DATA_BLOCK "LBP_SentronPac"   // DB1001
TITLE = SENTRON PAC
{ S7_Optimized_Access := 'FALSE'; DB_Accessible_From_OPC_UA := 'FALSE' }
AUTHOR : SINUMERIK
FAMILY : SINUMERIK_ONE
VERSION : 6.24
// Interface between user program and operating software, contains signals for SENTRON PAC energy monitoring devices / Interface entre programme utilisateur et logiciel d'exploitation, contient des signaux pour unités de surveillance de l'énergie SENTRON PAC
// stored: AutoNumber false, DBAccessibleFromOPCUA false, DBAccessibleFromWebserver false
   VAR RETAIN
      ManualVal { ExternalWritable := 'False'} : Bool;   // Display of manual value / Affichage de la valeur manuelle
      SentronPacMach { ExternalWritable := 'False'} : Bool;   // Sentron PAC represented machine / Machine représentée par Sentron PAC
      FeedInEnergyReadSP { ExternalWritable := 'False'} : Bool;   // Feed-in energy read from Sentron PAC / Énergie alimentée mesurée par Sentron PAC
      FeedBackEnergyReadSP { ExternalWritable := 'False'} : Bool;   // Feed back energy read from Sentron PAC / Énergie réinjectée mesurée par Sentron PAC
      FeedInEnergyReadAuxil { ExternalWritable := 'False'} : Bool;   // Feed-in energy read auxiliary / Énergie alimentée, mesurée par AUX
      FeedBackEnergyReadAuxil { ExternalWritable := 'False'} : Bool;   // Feed back energy read auxiliary / Énergie réinjectée, mesurée par AUX
      res0_6 { ExternalWritable := 'False'} : Bool;   // Reserved / Réservé
      res0_7 { ExternalWritable := 'False'} : Bool;   // Reserved / Réservé
      MeasAuto { ExternalWritable := 'False'} : Bool;   // Measurement by PLC basic program / Mesure par programme de base AP
      res1_1 { ExternalWritable := 'False'} : Bool;   // Reserved / Réservé
      res1_2 { ExternalWritable := 'False'} : Bool;   // Reserved / Réservé
      res1_3 { ExternalWritable := 'False'} : Bool;   // Reserved / Réservé
      res1_4 { ExternalWritable := 'False'} : Bool;   // Reserved / Réservé
      res1_5 { ExternalWritable := 'False'} : Bool;   // Reserved / Réservé
      res1_6 { ExternalWritable := 'False'} : Bool;   // Reserved / Réservé
      res1_7 { ExternalWritable := 'False'} : Bool;   // Reserved / Réservé
      MeasAct : Bool;   // HMI -> PLC: Active measurement / IHM->AP : Mesure active
      res2_1 { ExternalWritable := 'False'} : Bool;   // Reserved / Réservé
      res2_2 { ExternalWritable := 'False'} : Bool;   // Reserved / Réservé
      res2_3 { ExternalWritable := 'False'} : Bool;   // Reserved / Réservé
      res2_4 { ExternalWritable := 'False'} : Bool;   // Reserved / Réservé
      res2_5 { ExternalWritable := 'False'} : Bool;   // Reserved / Réservé
      res2_6 { ExternalWritable := 'False'} : Bool;   // Reserved / Réservé
      res2_7 { ExternalWritable := 'False'} : Bool;   // Reserved / Réservé
      EStateOn { ExternalWritable := 'False'} : Bool;   // Energy state on / État énergie activé
      res3_1 { ExternalWritable := 'False'} : Bool;   // Reserved / Réservé
      res3_2 { ExternalWritable := 'False'} : Bool;   // Reserved / Réservé
      res3_3 { ExternalWritable := 'False'} : Bool;   // Reserved / Réservé
      res3_4 { ExternalWritable := 'False'} : Bool;   // Reserved / Réservé
      res3_5 { ExternalWritable := 'False'} : Bool;   // Reserved / Réservé
      res3_6 { ExternalWritable := 'False'} : Bool;   // Reserved / Réservé
      res3_7 { ExternalWritable := 'False'} : Bool;   // Reserved / Réservé
      ManualValue { ExternalWritable := 'False'} : Real;   // Manual value / Valeur manuelle
      ActivePowerItem { ExternalWritable := 'False'} : Real;   // Active power item / Puissance active position
      ActiveEnergyItem { ExternalWritable := 'False'} : Real;   // Active energy item / Énergie active position
      ReactiveEnergyItem { ExternalWritable := 'False'} : Real;   // Reactive energy item / Énergie réactive position
      ActivePowerSentron { ExternalWritable := 'False'} : Real;   // Active power from Sentron / Puissance active par Sentron
      ActiveEnergySentron { ExternalWritable := 'False'} : Real;   // Active energy from Sentron / Énergie active par Sentron
      ReactiveEnergySentron { ExternalWritable := 'False'} : Real;   // Reactive energy from Sentron / Énergie réactive par Sentron
      ActiveEnergyDay { ExternalWritable := 'False'} : Real;   // Active energy day / Énergie active jour
      ReactiveEnergyDay { ExternalWritable := 'False'} : Real;   // Reactive energy day / Énergie réactive jour
      ActiveEnergyPrevDay { ExternalWritable := 'False'} : Real;   // Active energy previous day / Énergie active jour précédent
      ReactiveEnergyPrevDay { ExternalWritable := 'False'} : Real;   // Reactive energy previous day / Énergie réactive jour précédent
      ActiveEnergyMonth { ExternalWritable := 'False'} : Real;   // Active energy month / Énergie active mois
      ReactiveEnergyMonth { ExternalWritable := 'False'} : Real;   // Reactive energy month / Énergie réactive mois
      ActiveEnergyPrevMonth { ExternalWritable := 'False'} : Real;   // Active energy previous month / Énergie active mois précédent
      ReactiveEnergyPrevMonth { ExternalWritable := 'False'} : Real;   // Reactive energy previous month / Énergie réactive mois précédent
      ActiveEnergyYear { ExternalWritable := 'False'} : Real;   // Active energy year / Énergie active année
      ReactiveEnergyYear { ExternalWritable := 'False'} : Real;   // Reactive energy year / Énergie réactive année
      ActiveEnergyPrevYear { ExternalWritable := 'False'} : Real;   // Active energy previous year / Énergie active année précédente
      ReactiveEnergyPrevYear { ExternalWritable := 'False'} : Real;   // Reactive energy previous year / Énergie réactive année précédente
      res80 { ExternalWritable := 'False'} : Byte;   // Reserved / Réservé
      res81 { ExternalWritable := 'False'} : Byte;   // Reserved / Réservé
      res82 { ExternalWritable := 'False'} : Byte;   // Reserved / Réservé
      res83 { ExternalWritable := 'False'} : Byte;   // Reserved / Réservé
      res84 { ExternalWritable := 'False'} : Byte;   // Reserved / Réservé
      res85 { ExternalWritable := 'False'} : Byte;   // Reserved / Réservé
      res86 { ExternalWritable := 'False'} : Byte;   // Reserved / Réservé
      res87 { ExternalWritable := 'False'} : Byte;   // Reserved / Réservé
      res88 { ExternalWritable := 'False'} : Real;   // Reserved / Réservé
      res92 { ExternalWritable := 'False'} : Real;   // Reserved / Réservé
      ProductionAct { ExternalWritable := 'False'} : Byte;
      ErrDBD20_NAN { ExternalWritable := 'False'} : Bool;   // DBD20: invalid (not a number) / DBD20 : non valide (pas un nombre)
      ErrDBD24_NAN { ExternalWritable := 'False'} : Bool;   // DBD24: invalid (not a number) / DBD24 : non valide (pas un nombre)
      ErrDBD28_NAN { ExternalWritable := 'False'} : Bool;   // DBD28: invalid (not a number) / DBD28 : non valide (pas un nombre)
      res97_3 { ExternalWritable := 'False'} : Bool;   // Reserved / Réservé
      res97_4 { ExternalWritable := 'False'} : Bool;   // Reserved / Réservé
      res97_5 { ExternalWritable := 'False'} : Bool;   // Reserved / Réservé
      res97_6 { ExternalWritable := 'False'} : Bool;   // Reserved / Réservé
      res97_7 { ExternalWritable := 'False'} : Bool;   // Reserved / Réservé
      ErrDBD104_NAN { ExternalWritable := 'False'} : Bool;   // DBD104: invalid (not a number) / DBD104 : non valide (pas un nombre)
      ErrDBD144_NAN { ExternalWritable := 'False'} : Bool;   // DBD144: invalid (not a number) / DBD144 : non valide (pas un nombre)
      ErrDBD184_NAN { ExternalWritable := 'False'} : Bool;   // DBD184: invalid (not a number) / DBD184 : non valide (pas un nombre)
      ErrDBD224_NAN { ExternalWritable := 'False'} : Bool;   // DBD224: invalid (not a number) / DBD224 : non valide (pas un nombre)
      ErrDBD264_NAN { ExternalWritable := 'False'} : Bool;   // DBD264: invalid (not a number) / DBD264 : non valide (pas un nombre)
      ErrDBD304_NAN { ExternalWritable := 'False'} : Bool;   // DBD304: invalid (not a number) / DBD304 : non valide (pas un nombre)
      ErrDBD344_NAN { ExternalWritable := 'False'} : Bool;   // DBD344: invalid (not a number) / DBD344 : non valide (pas un nombre)
      ErrDBD384_NAN { ExternalWritable := 'False'} : Bool;   // DBD384: invalid (not a number) / DBD384 : non valide (pas un nombre)
      ErrDBD424_NAN { ExternalWritable := 'False'} : Bool;   // DBD424: invalid (not a number) / DBD424 : non valide (pas un nombre)
      ErrDBD464_NAN { ExternalWritable := 'False'} : Bool;   // DBD464: invalid (not a number) / DBD464 : non valide (pas un nombre)
      res99_2 { ExternalWritable := 'False'} : Bool;   // Reserved / Réservé
      res99_3 { ExternalWritable := 'False'} : Bool;   // Reserved / Réservé
      res99_4 { ExternalWritable := 'False'} : Bool;   // Reserved / Réservé
      res99_5 { ExternalWritable := 'False'} : Bool;   // Reserved / Réservé
      res99_6 { ExternalWritable := 'False'} : Bool;   // Reserved / Réservé
      res99_7 { ExternalWritable := 'False'} : Bool;   // Reserved / Réservé
      CtrlE_AuxDevice { ExternalWritable := 'False'} : Array[1..10] of Struct
         ProcessAux : Bool;   // Auxiliary present and to be processed / AUX présent et prêt au traitement
         ReadEnergy : Bool;   // Actual values are refreshed; bit is auto-reset / Les valeurs réelles sont actualisées ; le bit est réinitialisé automatiquement
         MeasAct : Bool;   // Measurement values are computed / Calcul des valeurs de mesure en cours
         MeasMode : Bool;   // Difference of actual values is stored / La différence des valeurs réelles est enregistrée
         InputMode : Bool;   // INPUT "ActivePowerAux" is energy in kWh / INPUT "ActivePowerAux" représente l'énergie en kWh
         res0_5 : Bool;
         res0_6 : Bool;
         ResetAux : Bool;   // Auxiliary data are deleted / Les données AUX sont supprimées
         res1 : Byte;   // Reserved / Réservé
         res2 : Word;   // Reserved / Réservé
         ActivePowerAux : Real;   // [kW]/[kWh] power/energy of auxiliary, written by customer / [kW]/[kWh] puissance/énergie AUX, renseignée par le client
         ActiveEnAux : Real;   // [kWh] actual value of fed-in-energy / [kWh] valeur réelle de l'énergie consommée
         ReActiveEnAux : Real;   // [kWh] actual value of fed-back energy / [kWh] valeur réelle de l'énergie réinjectée
         ActiveEnAuxMeasON : Real;   // [kWh] value of fed-in-energy at start of measurement / [kWh] valeur réelle de l'énergie consommée au début de la mesure
         ReActiveEnAuxMeasON : Real;   // [kWh] value of fed-back energy at start of measurement / Wh] valeur réelle de l'énergie réinjectée au début de la mesure
         ActiveEnAuxMeasOFF : Real;   // [kWh] value of fed-in-energy at end of measurement / [kWh] valeur réelle de l'énergie consommée à la fin de la mesure
         ReActiveEnAuxMeasOFF : Real;   // [kWh] value of fed-back energy at end of measurement / [kWh] valeur réelle de l'énergie réinjectée à la fin de la mesure
         res32 : DWord;   // Reserved / Réservé
         res36 : Real;   // Reserved / Réservé
      END_STRUCT;
   END_VAR
BEGIN
   // CtrlE_AuxDevice[2].ProcessAux : Auxiliary present and to be processed / AUX présent et prêt au traitement
   // CtrlE_AuxDevice[3].ProcessAux : Auxiliary present and to be processed / AUX présent et prêt au traitement
   // CtrlE_AuxDevice[4].ProcessAux : Auxiliary present and to be processed / AUX présent et prêt au traitement
   // CtrlE_AuxDevice[5].ProcessAux : Auxiliary present and to be processed / AUX présent et prêt au traitement
   // CtrlE_AuxDevice[6].ProcessAux : Auxiliary present and to be processed / AUX présent et prêt au traitement
   // CtrlE_AuxDevice[7].ProcessAux : Auxiliary present and to be processed / AUX présent et prêt au traitement
   // CtrlE_AuxDevice[8].ProcessAux : Auxiliary present and to be processed / AUX présent et prêt au traitement
   // CtrlE_AuxDevice[9].ProcessAux : Auxiliary present and to be processed / AUX présent et prêt au traitement
   // CtrlE_AuxDevice[10].ProcessAux : Auxiliary present and to be processed / AUX présent et prêt au traitement
   // CtrlE_AuxDevice[2].ReadEnergy : Actual values are refreshed; bit is auto-reset / Les valeurs réelles sont actualisées ; le bit est réinitialisé automatiquement
   // CtrlE_AuxDevice[3].ReadEnergy : Actual values are refreshed; bit is auto-reset / Les valeurs réelles sont actualisées ; le bit est réinitialisé automatiquement
   // CtrlE_AuxDevice[4].ReadEnergy : Actual values are refreshed; bit is auto-reset / Les valeurs réelles sont actualisées ; le bit est réinitialisé automatiquement
   // CtrlE_AuxDevice[5].ReadEnergy : Actual values are refreshed; bit is auto-reset / Les valeurs réelles sont actualisées ; le bit est réinitialisé automatiquement
   // CtrlE_AuxDevice[6].ReadEnergy : Actual values are refreshed; bit is auto-reset / Les valeurs réelles sont actualisées ; le bit est réinitialisé automatiquement
   // CtrlE_AuxDevice[7].ReadEnergy : Actual values are refreshed; bit is auto-reset / Les valeurs réelles sont actualisées ; le bit est réinitialisé automatiquement
   // CtrlE_AuxDevice[8].ReadEnergy : Actual values are refreshed; bit is auto-reset / Les valeurs réelles sont actualisées ; le bit est réinitialisé automatiquement
   // CtrlE_AuxDevice[9].ReadEnergy : Actual values are refreshed; bit is auto-reset / Les valeurs réelles sont actualisées ; le bit est réinitialisé automatiquement
   // CtrlE_AuxDevice[10].ReadEnergy : Actual values are refreshed; bit is auto-reset / Les valeurs réelles sont actualisées ; le bit est réinitialisé automatiquement
   // CtrlE_AuxDevice[2].MeasAct : Measurement values are computed / Calcul des valeurs de mesure en cours
   // CtrlE_AuxDevice[3].MeasAct : Measurement values are computed / Calcul des valeurs de mesure en cours
   // CtrlE_AuxDevice[4].MeasAct : Measurement values are computed / Calcul des valeurs de mesure en cours
   // CtrlE_AuxDevice[5].MeasAct : Measurement values are computed / Calcul des valeurs de mesure en cours
   // CtrlE_AuxDevice[6].MeasAct : Measurement values are computed / Calcul des valeurs de mesure en cours
   // CtrlE_AuxDevice[7].MeasAct : Measurement values are computed / Calcul des valeurs de mesure en cours
   // CtrlE_AuxDevice[8].MeasAct : Measurement values are computed / Calcul des valeurs de mesure en cours
   // CtrlE_AuxDevice[9].MeasAct : Measurement values are computed / Calcul des valeurs de mesure en cours
   // CtrlE_AuxDevice[10].MeasAct : Measurement values are computed / Calcul des valeurs de mesure en cours
   // CtrlE_AuxDevice[2].MeasMode : Difference of actual values is stored / La différence des valeurs réelles est enregistrée
   // CtrlE_AuxDevice[3].MeasMode : Difference of actual values is stored / La différence des valeurs réelles est enregistrée
   // CtrlE_AuxDevice[4].MeasMode : Difference of actual values is stored / La différence des valeurs réelles est enregistrée
   // CtrlE_AuxDevice[5].MeasMode : Difference of actual values is stored / La différence des valeurs réelles est enregistrée
   // CtrlE_AuxDevice[6].MeasMode : Difference of actual values is stored / La différence des valeurs réelles est enregistrée
   // CtrlE_AuxDevice[7].MeasMode : Difference of actual values is stored / La différence des valeurs réelles est enregistrée
   // CtrlE_AuxDevice[8].MeasMode : Difference of actual values is stored / La différence des valeurs réelles est enregistrée
   // CtrlE_AuxDevice[9].MeasMode : Difference of actual values is stored / La différence des valeurs réelles est enregistrée
   // CtrlE_AuxDevice[10].MeasMode : Difference of actual values is stored / La différence des valeurs réelles est enregistrée
   // CtrlE_AuxDevice[2].InputMode : INPUT "ActivePowerAux" is energy in kWh / INPUT "ActivePowerAux" représente l'énergie en kWh
   // CtrlE_AuxDevice[3].InputMode : INPUT "ActivePowerAux" is energy in kWh / INPUT "ActivePowerAux" représente l'énergie en kWh
   // CtrlE_AuxDevice[4].InputMode : INPUT "ActivePowerAux" is energy in kWh / INPUT "ActivePowerAux" représente l'énergie en kWh
   // CtrlE_AuxDevice[5].InputMode : INPUT "ActivePowerAux" is energy in kWh / INPUT "ActivePowerAux" représente l'énergie en kWh
   // CtrlE_AuxDevice[6].InputMode : INPUT "ActivePowerAux" is energy in kWh / INPUT "ActivePowerAux" représente l'énergie en kWh
   // CtrlE_AuxDevice[7].InputMode : INPUT "ActivePowerAux" is energy in kWh / INPUT "ActivePowerAux" représente l'énergie en kWh
   // CtrlE_AuxDevice[8].InputMode : INPUT "ActivePowerAux" is energy in kWh / INPUT "ActivePowerAux" représente l'énergie en kWh
   // CtrlE_AuxDevice[9].InputMode : INPUT "ActivePowerAux" is energy in kWh / INPUT "ActivePowerAux" représente l'énergie en kWh
   // CtrlE_AuxDevice[10].InputMode : INPUT "ActivePowerAux" is energy in kWh / INPUT "ActivePowerAux" représente l'énergie en kWh
   // CtrlE_AuxDevice[2].ResetAux : Auxiliary data are deleted / Les données AUX sont supprimées
   // CtrlE_AuxDevice[3].ResetAux : Auxiliary data are deleted / Les données AUX sont supprimées
   // CtrlE_AuxDevice[4].ResetAux : Auxiliary data are deleted / Les données AUX sont supprimées
   // CtrlE_AuxDevice[5].ResetAux : Auxiliary data are deleted / Les données AUX sont supprimées
   // CtrlE_AuxDevice[6].ResetAux : Auxiliary data are deleted / Les données AUX sont supprimées
   // CtrlE_AuxDevice[7].ResetAux : Auxiliary data are deleted / Les données AUX sont supprimées
   // CtrlE_AuxDevice[8].ResetAux : Auxiliary data are deleted / Les données AUX sont supprimées
   // CtrlE_AuxDevice[9].ResetAux : Auxiliary data are deleted / Les données AUX sont supprimées
   // CtrlE_AuxDevice[10].ResetAux : Auxiliary data are deleted / Les données AUX sont supprimées
   // CtrlE_AuxDevice[2].res1 : Reserved / Réservé
   // CtrlE_AuxDevice[3].res1 : Reserved / Réservé
   // CtrlE_AuxDevice[4].res1 : Reserved / Réservé
   // CtrlE_AuxDevice[5].res1 : Reserved / Réservé
   // CtrlE_AuxDevice[6].res1 : Reserved / Réservé
   // CtrlE_AuxDevice[7].res1 : Reserved / Réservé
   // CtrlE_AuxDevice[8].res1 : Reserved / Réservé
   // CtrlE_AuxDevice[9].res1 : Reserved / Réservé
   // CtrlE_AuxDevice[10].res1 : Reserved / Réservé
   // CtrlE_AuxDevice[2].res2 : Reserved / Réservé
   // CtrlE_AuxDevice[3].res2 : Reserved / Réservé
   // CtrlE_AuxDevice[4].res2 : Reserved / Réservé
   // CtrlE_AuxDevice[5].res2 : Reserved / Réservé
   // CtrlE_AuxDevice[6].res2 : Reserved / Réservé
   // CtrlE_AuxDevice[7].res2 : Reserved / Réservé
   // CtrlE_AuxDevice[8].res2 : Reserved / Réservé
   // CtrlE_AuxDevice[9].res2 : Reserved / Réservé
   // CtrlE_AuxDevice[10].res2 : Reserved / Réservé
   // CtrlE_AuxDevice[2].ActivePowerAux : [kW]/[kWh] power/energy of auxiliary, written by customer / [kW]/[kWh] puissance/énergie AUX, renseignée par le client
   // CtrlE_AuxDevice[3].ActivePowerAux : [kW]/[kWh] power/energy of auxiliary, written by customer / [kW]/[kWh] puissance/énergie AUX, renseignée par le client
   // CtrlE_AuxDevice[4].ActivePowerAux : [kW]/[kWh] power/energy of auxiliary, written by customer / [kW]/[kWh] puissance/énergie AUX, renseignée par le client
   // CtrlE_AuxDevice[5].ActivePowerAux : [kW]/[kWh] power/energy of auxiliary, written by customer / [kW]/[kWh] puissance/énergie AUX, renseignée par le client
   // CtrlE_AuxDevice[6].ActivePowerAux : [kW]/[kWh] power/energy of auxiliary, written by customer / [kW]/[kWh] puissance/énergie AUX, renseignée par le client
   // CtrlE_AuxDevice[7].ActivePowerAux : [kW]/[kWh] power/energy of auxiliary, written by customer / [kW]/[kWh] puissance/énergie AUX, renseignée par le client
   // CtrlE_AuxDevice[8].ActivePowerAux : [kW]/[kWh] power/energy of auxiliary, written by customer / [kW]/[kWh] puissance/énergie AUX, renseignée par le client
   // CtrlE_AuxDevice[9].ActivePowerAux : [kW]/[kWh] power/energy of auxiliary, written by customer / [kW]/[kWh] puissance/énergie AUX, renseignée par le client
   // CtrlE_AuxDevice[10].ActivePowerAux : [kW]/[kWh] power/energy of auxiliary, written by customer / [kW]/[kWh] puissance/énergie AUX, renseignée par le client
   // CtrlE_AuxDevice[2].ActiveEnAux : [kWh] actual value of fed-in-energy / [kWh] valeur réelle de l'énergie consommée
   // CtrlE_AuxDevice[3].ActiveEnAux : [kWh] actual value of fed-in-energy / [kWh] valeur réelle de l'énergie consommée
   // CtrlE_AuxDevice[4].ActiveEnAux : [kWh] actual value of fed-in-energy / [kWh] valeur réelle de l'énergie consommée
   // CtrlE_AuxDevice[5].ActiveEnAux : [kWh] actual value of fed-in-energy / [kWh] valeur réelle de l'énergie consommée
   // CtrlE_AuxDevice[6].ActiveEnAux : [kWh] actual value of fed-in-energy / [kWh] valeur réelle de l'énergie consommée
   // CtrlE_AuxDevice[7].ActiveEnAux : [kWh] actual value of fed-in-energy / [kWh] valeur réelle de l'énergie consommée
   // CtrlE_AuxDevice[8].ActiveEnAux : [kWh] actual value of fed-in-energy / [kWh] valeur réelle de l'énergie consommée
   // CtrlE_AuxDevice[9].ActiveEnAux : [kWh] actual value of fed-in-energy / [kWh] valeur réelle de l'énergie consommée
   // CtrlE_AuxDevice[10].ActiveEnAux : [kWh] actual value of fed-in-energy / [kWh] valeur réelle de l'énergie consommée
   // CtrlE_AuxDevice[2].ReActiveEnAux : [kWh] actual value of fed-back energy / [kWh] valeur réelle de l'énergie réinjectée
   // CtrlE_AuxDevice[3].ReActiveEnAux : [kWh] actual value of fed-back energy / [kWh] valeur réelle de l'énergie réinjectée
   // CtrlE_AuxDevice[4].ReActiveEnAux : [kWh] actual value of fed-back energy / [kWh] valeur réelle de l'énergie réinjectée
   // CtrlE_AuxDevice[5].ReActiveEnAux : [kWh] actual value of fed-back energy / [kWh] valeur réelle de l'énergie réinjectée
   // CtrlE_AuxDevice[6].ReActiveEnAux : [kWh] actual value of fed-back energy / [kWh] valeur réelle de l'énergie réinjectée
   // CtrlE_AuxDevice[7].ReActiveEnAux : [kWh] actual value of fed-back energy / [kWh] valeur réelle de l'énergie réinjectée
   // CtrlE_AuxDevice[8].ReActiveEnAux : [kWh] actual value of fed-back energy / [kWh] valeur réelle de l'énergie réinjectée
   // CtrlE_AuxDevice[9].ReActiveEnAux : [kWh] actual value of fed-back energy / [kWh] valeur réelle de l'énergie réinjectée
   // CtrlE_AuxDevice[10].ReActiveEnAux : [kWh] actual value of fed-back energy / [kWh] valeur réelle de l'énergie réinjectée
   // CtrlE_AuxDevice[2].ActiveEnAuxMeasON : [kWh] value of fed-in-energy at start of measurement / [kWh] valeur réelle de l'énergie consommée au début de la mesure
   // CtrlE_AuxDevice[3].ActiveEnAuxMeasON : [kWh] value of fed-in-energy at start of measurement / [kWh] valeur réelle de l'énergie consommée au début de la mesure
   // CtrlE_AuxDevice[4].ActiveEnAuxMeasON : [kWh] value of fed-in-energy at start of measurement / [kWh] valeur réelle de l'énergie consommée au début de la mesure
   // CtrlE_AuxDevice[5].ActiveEnAuxMeasON : [kWh] value of fed-in-energy at start of measurement / [kWh] valeur réelle de l'énergie consommée au début de la mesure
   // CtrlE_AuxDevice[6].ActiveEnAuxMeasON : [kWh] value of fed-in-energy at start of measurement / [kWh] valeur réelle de l'énergie consommée au début de la mesure
   // CtrlE_AuxDevice[7].ActiveEnAuxMeasON : [kWh] value of fed-in-energy at start of measurement / [kWh] valeur réelle de l'énergie consommée au début de la mesure
   // CtrlE_AuxDevice[8].ActiveEnAuxMeasON : [kWh] value of fed-in-energy at start of measurement / [kWh] valeur réelle de l'énergie consommée au début de la mesure
   // CtrlE_AuxDevice[9].ActiveEnAuxMeasON : [kWh] value of fed-in-energy at start of measurement / [kWh] valeur réelle de l'énergie consommée au début de la mesure
   // CtrlE_AuxDevice[10].ActiveEnAuxMeasON : [kWh] value of fed-in-energy at start of measurement / [kWh] valeur réelle de l'énergie consommée au début de la mesure
   // CtrlE_AuxDevice[2].ReActiveEnAuxMeasON : [kWh] value of fed-back energy at start of measurement / Wh] valeur réelle de l'énergie réinjectée au début de la mesure
   // CtrlE_AuxDevice[3].ReActiveEnAuxMeasON : [kWh] value of fed-back energy at start of measurement / Wh] valeur réelle de l'énergie réinjectée au début de la mesure
   // CtrlE_AuxDevice[4].ReActiveEnAuxMeasON : [kWh] value of fed-back energy at start of measurement / Wh] valeur réelle de l'énergie réinjectée au début de la mesure
   // CtrlE_AuxDevice[5].ReActiveEnAuxMeasON : [kWh] value of fed-back energy at start of measurement / Wh] valeur réelle de l'énergie réinjectée au début de la mesure
   // CtrlE_AuxDevice[6].ReActiveEnAuxMeasON : [kWh] value of fed-back energy at start of measurement / Wh] valeur réelle de l'énergie réinjectée au début de la mesure
   // CtrlE_AuxDevice[7].ReActiveEnAuxMeasON : [kWh] value of fed-back energy at start of measurement / Wh] valeur réelle de l'énergie réinjectée au début de la mesure
   // CtrlE_AuxDevice[8].ReActiveEnAuxMeasON : [kWh] value of fed-back energy at start of measurement / Wh] valeur réelle de l'énergie réinjectée au début de la mesure
   // CtrlE_AuxDevice[9].ReActiveEnAuxMeasON : [kWh] value of fed-back energy at start of measurement / Wh] valeur réelle de l'énergie réinjectée au début de la mesure
   // CtrlE_AuxDevice[10].ReActiveEnAuxMeasON : [kWh] value of fed-back energy at start of measurement / Wh] valeur réelle de l'énergie réinjectée au début de la mesure
   // CtrlE_AuxDevice[2].ActiveEnAuxMeasOFF : [kWh] value of fed-in-energy at end of measurement / [kWh] valeur réelle de l'énergie consommée à la fin de la mesure
   // CtrlE_AuxDevice[3].ActiveEnAuxMeasOFF : [kWh] value of fed-in-energy at end of measurement / [kWh] valeur réelle de l'énergie consommée à la fin de la mesure
   // CtrlE_AuxDevice[4].ActiveEnAuxMeasOFF : [kWh] value of fed-in-energy at end of measurement / [kWh] valeur réelle de l'énergie consommée à la fin de la mesure
   // CtrlE_AuxDevice[5].ActiveEnAuxMeasOFF : [kWh] value of fed-in-energy at end of measurement / [kWh] valeur réelle de l'énergie consommée à la fin de la mesure
   // CtrlE_AuxDevice[6].ActiveEnAuxMeasOFF : [kWh] value of fed-in-energy at end of measurement / [kWh] valeur réelle de l'énergie consommée à la fin de la mesure
   // CtrlE_AuxDevice[7].ActiveEnAuxMeasOFF : [kWh] value of fed-in-energy at end of measurement / [kWh] valeur réelle de l'énergie consommée à la fin de la mesure
   // CtrlE_AuxDevice[8].ActiveEnAuxMeasOFF : [kWh] value of fed-in-energy at end of measurement / [kWh] valeur réelle de l'énergie consommée à la fin de la mesure
   // CtrlE_AuxDevice[9].ActiveEnAuxMeasOFF : [kWh] value of fed-in-energy at end of measurement / [kWh] valeur réelle de l'énergie consommée à la fin de la mesure
   // CtrlE_AuxDevice[10].ActiveEnAuxMeasOFF : [kWh] value of fed-in-energy at end of measurement / [kWh] valeur réelle de l'énergie consommée à la fin de la mesure
   // CtrlE_AuxDevice[2].ReActiveEnAuxMeasOFF : [kWh] value of fed-back energy at end of measurement / [kWh] valeur réelle de l'énergie réinjectée à la fin de la mesure
   // CtrlE_AuxDevice[3].ReActiveEnAuxMeasOFF : [kWh] value of fed-back energy at end of measurement / [kWh] valeur réelle de l'énergie réinjectée à la fin de la mesure
   // CtrlE_AuxDevice[4].ReActiveEnAuxMeasOFF : [kWh] value of fed-back energy at end of measurement / [kWh] valeur réelle de l'énergie réinjectée à la fin de la mesure
   // CtrlE_AuxDevice[5].ReActiveEnAuxMeasOFF : [kWh] value of fed-back energy at end of measurement / [kWh] valeur réelle de l'énergie réinjectée à la fin de la mesure
   // CtrlE_AuxDevice[6].ReActiveEnAuxMeasOFF : [kWh] value of fed-back energy at end of measurement / [kWh] valeur réelle de l'énergie réinjectée à la fin de la mesure
   // CtrlE_AuxDevice[7].ReActiveEnAuxMeasOFF : [kWh] value of fed-back energy at end of measurement / [kWh] valeur réelle de l'énergie réinjectée à la fin de la mesure
   // CtrlE_AuxDevice[8].ReActiveEnAuxMeasOFF : [kWh] value of fed-back energy at end of measurement / [kWh] valeur réelle de l'énergie réinjectée à la fin de la mesure
   // CtrlE_AuxDevice[9].ReActiveEnAuxMeasOFF : [kWh] value of fed-back energy at end of measurement / [kWh] valeur réelle de l'énergie réinjectée à la fin de la mesure
   // CtrlE_AuxDevice[10].ReActiveEnAuxMeasOFF : [kWh] value of fed-back energy at end of measurement / [kWh] valeur réelle de l'énergie réinjectée à la fin de la mesure
   // CtrlE_AuxDevice[2].res32 : Reserved / Réservé
   // CtrlE_AuxDevice[3].res32 : Reserved / Réservé
   // CtrlE_AuxDevice[4].res32 : Reserved / Réservé
   // CtrlE_AuxDevice[5].res32 : Reserved / Réservé
   // CtrlE_AuxDevice[6].res32 : Reserved / Réservé
   // CtrlE_AuxDevice[7].res32 : Reserved / Réservé
   // CtrlE_AuxDevice[8].res32 : Reserved / Réservé
   // CtrlE_AuxDevice[9].res32 : Reserved / Réservé
   // CtrlE_AuxDevice[10].res32 : Reserved / Réservé
   // CtrlE_AuxDevice[2].res36 : Reserved / Réservé
   // CtrlE_AuxDevice[3].res36 : Reserved / Réservé
   // CtrlE_AuxDevice[4].res36 : Reserved / Réservé
   // CtrlE_AuxDevice[5].res36 : Reserved / Réservé
   // CtrlE_AuxDevice[6].res36 : Reserved / Réservé
   // CtrlE_AuxDevice[7].res36 : Reserved / Réservé
   // CtrlE_AuxDevice[8].res36 : Reserved / Réservé
   // CtrlE_AuxDevice[9].res36 : Reserved / Réservé
   // CtrlE_AuxDevice[10].res36 : Reserved / Réservé
END_DATA_BLOCK

DATA_BLOCK "LBP_SpindleTempSensor"   // DB1002
TITLE = Spindle temperature sensors / Sondes thermométriques de broche
{ S7_Optimized_Access := 'FALSE' }
AUTHOR : SINUMERIK
FAMILY : SINUMERIK_ONE
VERSION : 6.24
// Interface between user program and operating software, contains signals for spindle temperature sensors / Interface entre programme utilisateur et logiciel d'exploitation, contient des signaux pour sondes thermométriques de broche
// stored: AutoNumber false
   VAR RETAIN
      Sp : Array[1..2] of Struct   // Spindle / Broche
         TS : Array[1..6] of Struct   // Temperature sensor / Sonde thermométrique
            MountPlace : Int;   // Sensor assembly location / Emplacement du module capteur
            Res1 : Int;
            ActVal : Real;   // Temperature sensor actual value [°C] / Sonde thermométrique valeur réelle [°C]
            WarnThreshold : Real;   // Temperature sensor warning threshold value [°C] / Sonde thermométrique valeur seuil d'alarme
            WarnNumLimitViol : Int;   // Number of warning threshold value violations / Nombre de dépassements de la valeur seuil d'alarme
            WarnTsViolYY : Byte;   // Last warning threshold value violation: year / Dernier dépassement de la valeur seuil d'alarme : année
            WarnTsViolMM : Byte;   // Last warning threshold value violation: month / Dernier dépassement de la valeur seuil d'alarme : mois
            WarnTsViolDD : Byte;   // Last warning threshold value violation: day / Dernier dépassement de la valeur seuil d'alarme : jour
            WarnTsViolH : Byte;   // Last warning threshold value violation: hour / Dernier dépassement de la valeur seuil d'alarme : heure
            WarnTsViolM : Byte;   // Last warning threshold value violation: minute / Dernier dépassement de la valeur seuil d'alarme : minute
            WarnTsViolS : Byte;   // Last warning threshold value violation: second / Dernier dépassement de la valeur seuil d'alarme : seconde
            WarnDurLimitViol : DInt;   // Duration of warning threshold value violations / Durée de dépassement de la valeur seuil d'alarme
            FaultThreshold : Real;   // Temperature sensor fault threshold value [°C] / Sonde thermométrique valeur seuil de défaut
            FaultNumLimitViol : Int;   // Number of fault threshold value violations / Nombre de dépassements de la valeur seuil de défaut
            FaultTsViolYY : Byte;   // Last fault threshold value violation: year / Dernier dépassement de la valeur seuil de défaut : année
            FaultTsViolMM : Byte;   // Last fault threshold value violation: month / Dernier dépassement de la valeur seuil de défaut : mois
            FaultTsViolDD : Byte;   // Last fault threshold value violation: day / Dernier dépassement de la valeur seuil de défaut : jour
            FaultTsViolH : Byte;   // Last fault threshold value violation: hour / Dernier dépassement de la valeur seuil de défaut : heure
            FaultTsViolM : Byte;   // Last fault threshold value violation: minute / Dernier dépassement de la valeur seuil de défaut : minute
            FaultTsViolS : Byte;   // Last fault threshold value violation: second / Dernier dépassement de la valeur seuil de défaut : seconde
            FaultDurLimitViol : DInt;   // Duration of fault threshold value violations / Durée de dépassement de la valeur seuil de défaut
         END_STRUCT;
      END_STRUCT;
   END_VAR
BEGIN
   // Sp[1].TS[2].MountPlace : Sensor assembly location / Emplacement du module capteur
   // Sp[1].TS[3].MountPlace : Sensor assembly location / Emplacement du module capteur
   // Sp[1].TS[4].MountPlace : Sensor assembly location / Emplacement du module capteur
   // Sp[1].TS[5].MountPlace : Sensor assembly location / Emplacement du module capteur
   // Sp[1].TS[6].MountPlace : Sensor assembly location / Emplacement du module capteur
   // Sp[2].TS[1].MountPlace : Sensor assembly location / Emplacement du module capteur
   // Sp[2].TS[2].MountPlace : Sensor assembly location / Emplacement du module capteur
   // Sp[2].TS[3].MountPlace : Sensor assembly location / Emplacement du module capteur
   // Sp[2].TS[4].MountPlace : Sensor assembly location / Emplacement du module capteur
   // Sp[2].TS[5].MountPlace : Sensor assembly location / Emplacement du module capteur
   // Sp[2].TS[6].MountPlace : Sensor assembly location / Emplacement du module capteur
   // Sp[1].TS[2].ActVal : Temperature sensor actual value [°C] / Sonde thermométrique valeur réelle [°C]
   // Sp[1].TS[3].ActVal : Temperature sensor actual value [°C] / Sonde thermométrique valeur réelle [°C]
   // Sp[1].TS[4].ActVal : Temperature sensor actual value [°C] / Sonde thermométrique valeur réelle [°C]
   // Sp[1].TS[5].ActVal : Temperature sensor actual value [°C] / Sonde thermométrique valeur réelle [°C]
   // Sp[1].TS[6].ActVal : Temperature sensor actual value [°C] / Sonde thermométrique valeur réelle [°C]
   // Sp[2].TS[1].ActVal : Temperature sensor actual value [°C] / Sonde thermométrique valeur réelle [°C]
   // Sp[2].TS[2].ActVal : Temperature sensor actual value [°C] / Sonde thermométrique valeur réelle [°C]
   // Sp[2].TS[3].ActVal : Temperature sensor actual value [°C] / Sonde thermométrique valeur réelle [°C]
   // Sp[2].TS[4].ActVal : Temperature sensor actual value [°C] / Sonde thermométrique valeur réelle [°C]
   // Sp[2].TS[5].ActVal : Temperature sensor actual value [°C] / Sonde thermométrique valeur réelle [°C]
   // Sp[2].TS[6].ActVal : Temperature sensor actual value [°C] / Sonde thermométrique valeur réelle [°C]
   // Sp[1].TS[2].WarnThreshold : Temperature sensor warning threshold value [°C] / Sonde thermométrique valeur seuil d'alarme
   // Sp[1].TS[3].WarnThreshold : Temperature sensor warning threshold value [°C] / Sonde thermométrique valeur seuil d'alarme
   // Sp[1].TS[4].WarnThreshold : Temperature sensor warning threshold value [°C] / Sonde thermométrique valeur seuil d'alarme
   // Sp[1].TS[5].WarnThreshold : Temperature sensor warning threshold value [°C] / Sonde thermométrique valeur seuil d'alarme
   // Sp[1].TS[6].WarnThreshold : Temperature sensor warning threshold value [°C] / Sonde thermométrique valeur seuil d'alarme
   // Sp[2].TS[1].WarnThreshold : Temperature sensor warning threshold value [°C] / Sonde thermométrique valeur seuil d'alarme
   // Sp[2].TS[2].WarnThreshold : Temperature sensor warning threshold value [°C] / Sonde thermométrique valeur seuil d'alarme
   // Sp[2].TS[3].WarnThreshold : Temperature sensor warning threshold value [°C] / Sonde thermométrique valeur seuil d'alarme
   // Sp[2].TS[4].WarnThreshold : Temperature sensor warning threshold value [°C] / Sonde thermométrique valeur seuil d'alarme
   // Sp[2].TS[5].WarnThreshold : Temperature sensor warning threshold value [°C] / Sonde thermométrique valeur seuil d'alarme
   // Sp[2].TS[6].WarnThreshold : Temperature sensor warning threshold value [°C] / Sonde thermométrique valeur seuil d'alarme
   // Sp[1].TS[2].WarnNumLimitViol : Number of warning threshold value violations / Nombre de dépassements de la valeur seuil d'alarme
   // Sp[1].TS[3].WarnNumLimitViol : Number of warning threshold value violations / Nombre de dépassements de la valeur seuil d'alarme
   // Sp[1].TS[4].WarnNumLimitViol : Number of warning threshold value violations / Nombre de dépassements de la valeur seuil d'alarme
   // Sp[1].TS[5].WarnNumLimitViol : Number of warning threshold value violations / Nombre de dépassements de la valeur seuil d'alarme
   // Sp[1].TS[6].WarnNumLimitViol : Number of warning threshold value violations / Nombre de dépassements de la valeur seuil d'alarme
   // Sp[2].TS[1].WarnNumLimitViol : Number of warning threshold value violations / Nombre de dépassements de la valeur seuil d'alarme
   // Sp[2].TS[2].WarnNumLimitViol : Number of warning threshold value violations / Nombre de dépassements de la valeur seuil d'alarme
   // Sp[2].TS[3].WarnNumLimitViol : Number of warning threshold value violations / Nombre de dépassements de la valeur seuil d'alarme
   // Sp[2].TS[4].WarnNumLimitViol : Number of warning threshold value violations / Nombre de dépassements de la valeur seuil d'alarme
   // Sp[2].TS[5].WarnNumLimitViol : Number of warning threshold value violations / Nombre de dépassements de la valeur seuil d'alarme
   // Sp[2].TS[6].WarnNumLimitViol : Number of warning threshold value violations / Nombre de dépassements de la valeur seuil d'alarme
   // Sp[1].TS[2].WarnTsViolYY : Last warning threshold value violation: year / Dernier dépassement de la valeur seuil d'alarme : année
   // Sp[1].TS[3].WarnTsViolYY : Last warning threshold value violation: year / Dernier dépassement de la valeur seuil d'alarme : année
   // Sp[1].TS[4].WarnTsViolYY : Last warning threshold value violation: year / Dernier dépassement de la valeur seuil d'alarme : année
   // Sp[1].TS[5].WarnTsViolYY : Last warning threshold value violation: year / Dernier dépassement de la valeur seuil d'alarme : année
   // Sp[1].TS[6].WarnTsViolYY : Last warning threshold value violation: year / Dernier dépassement de la valeur seuil d'alarme : année
   // Sp[2].TS[1].WarnTsViolYY : Last warning threshold value violation: year / Dernier dépassement de la valeur seuil d'alarme : année
   // Sp[2].TS[2].WarnTsViolYY : Last warning threshold value violation: year / Dernier dépassement de la valeur seuil d'alarme : année
   // Sp[2].TS[3].WarnTsViolYY : Last warning threshold value violation: year / Dernier dépassement de la valeur seuil d'alarme : année
   // Sp[2].TS[4].WarnTsViolYY : Last warning threshold value violation: year / Dernier dépassement de la valeur seuil d'alarme : année
   // Sp[2].TS[5].WarnTsViolYY : Last warning threshold value violation: year / Dernier dépassement de la valeur seuil d'alarme : année
   // Sp[2].TS[6].WarnTsViolYY : Last warning threshold value violation: year / Dernier dépassement de la valeur seuil d'alarme : année
   // Sp[1].TS[2].WarnTsViolMM : Last warning threshold value violation: month / Dernier dépassement de la valeur seuil d'alarme : mois
   // Sp[1].TS[3].WarnTsViolMM : Last warning threshold value violation: month / Dernier dépassement de la valeur seuil d'alarme : mois
   // Sp[1].TS[4].WarnTsViolMM : Last warning threshold value violation: month / Dernier dépassement de la valeur seuil d'alarme : mois
   // Sp[1].TS[5].WarnTsViolMM : Last warning threshold value violation: month / Dernier dépassement de la valeur seuil d'alarme : mois
   // Sp[1].TS[6].WarnTsViolMM : Last warning threshold value violation: month / Dernier dépassement de la valeur seuil d'alarme : mois
   // Sp[2].TS[1].WarnTsViolMM : Last warning threshold value violation: month / Dernier dépassement de la valeur seuil d'alarme : mois
   // Sp[2].TS[2].WarnTsViolMM : Last warning threshold value violation: month / Dernier dépassement de la valeur seuil d'alarme : mois
   // Sp[2].TS[3].WarnTsViolMM : Last warning threshold value violation: month / Dernier dépassement de la valeur seuil d'alarme : mois
   // Sp[2].TS[4].WarnTsViolMM : Last warning threshold value violation: month / Dernier dépassement de la valeur seuil d'alarme : mois
   // Sp[2].TS[5].WarnTsViolMM : Last warning threshold value violation: month / Dernier dépassement de la valeur seuil d'alarme : mois
   // Sp[2].TS[6].WarnTsViolMM : Last warning threshold value violation: month / Dernier dépassement de la valeur seuil d'alarme : mois
   // Sp[1].TS[2].WarnTsViolDD : Last warning threshold value violation: day / Dernier dépassement de la valeur seuil d'alarme : jour
   // Sp[1].TS[3].WarnTsViolDD : Last warning threshold value violation: day / Dernier dépassement de la valeur seuil d'alarme : jour
   // Sp[1].TS[4].WarnTsViolDD : Last warning threshold value violation: day / Dernier dépassement de la valeur seuil d'alarme : jour
   // Sp[1].TS[5].WarnTsViolDD : Last warning threshold value violation: day / Dernier dépassement de la valeur seuil d'alarme : jour
   // Sp[1].TS[6].WarnTsViolDD : Last warning threshold value violation: day / Dernier dépassement de la valeur seuil d'alarme : jour
   // Sp[2].TS[1].WarnTsViolDD : Last warning threshold value violation: day / Dernier dépassement de la valeur seuil d'alarme : jour
   // Sp[2].TS[2].WarnTsViolDD : Last warning threshold value violation: day / Dernier dépassement de la valeur seuil d'alarme : jour
   // Sp[2].TS[3].WarnTsViolDD : Last warning threshold value violation: day / Dernier dépassement de la valeur seuil d'alarme : jour
   // Sp[2].TS[4].WarnTsViolDD : Last warning threshold value violation: day / Dernier dépassement de la valeur seuil d'alarme : jour
   // Sp[2].TS[5].WarnTsViolDD : Last warning threshold value violation: day / Dernier dépassement de la valeur seuil d'alarme : jour
   // Sp[2].TS[6].WarnTsViolDD : Last warning threshold value violation: day / Dernier dépassement de la valeur seuil d'alarme : jour
   // Sp[1].TS[2].WarnTsViolH : Last warning threshold value violation: hour / Dernier dépassement de la valeur seuil d'alarme : heure
   // Sp[1].TS[3].WarnTsViolH : Last warning threshold value violation: hour / Dernier dépassement de la valeur seuil d'alarme : heure
   // Sp[1].TS[4].WarnTsViolH : Last warning threshold value violation: hour / Dernier dépassement de la valeur seuil d'alarme : heure
   // Sp[1].TS[5].WarnTsViolH : Last warning threshold value violation: hour / Dernier dépassement de la valeur seuil d'alarme : heure
   // Sp[1].TS[6].WarnTsViolH : Last warning threshold value violation: hour / Dernier dépassement de la valeur seuil d'alarme : heure
   // Sp[2].TS[1].WarnTsViolH : Last warning threshold value violation: hour / Dernier dépassement de la valeur seuil d'alarme : heure
   // Sp[2].TS[2].WarnTsViolH : Last warning threshold value violation: hour / Dernier dépassement de la valeur seuil d'alarme : heure
   // Sp[2].TS[3].WarnTsViolH : Last warning threshold value violation: hour / Dernier dépassement de la valeur seuil d'alarme : heure
   // Sp[2].TS[4].WarnTsViolH : Last warning threshold value violation: hour / Dernier dépassement de la valeur seuil d'alarme : heure
   // Sp[2].TS[5].WarnTsViolH : Last warning threshold value violation: hour / Dernier dépassement de la valeur seuil d'alarme : heure
   // Sp[2].TS[6].WarnTsViolH : Last warning threshold value violation: hour / Dernier dépassement de la valeur seuil d'alarme : heure
   // Sp[1].TS[2].WarnTsViolM : Last warning threshold value violation: minute / Dernier dépassement de la valeur seuil d'alarme : minute
   // Sp[1].TS[3].WarnTsViolM : Last warning threshold value violation: minute / Dernier dépassement de la valeur seuil d'alarme : minute
   // Sp[1].TS[4].WarnTsViolM : Last warning threshold value violation: minute / Dernier dépassement de la valeur seuil d'alarme : minute
   // Sp[1].TS[5].WarnTsViolM : Last warning threshold value violation: minute / Dernier dépassement de la valeur seuil d'alarme : minute
   // Sp[1].TS[6].WarnTsViolM : Last warning threshold value violation: minute / Dernier dépassement de la valeur seuil d'alarme : minute
   // Sp[2].TS[1].WarnTsViolM : Last warning threshold value violation: minute / Dernier dépassement de la valeur seuil d'alarme : minute
   // Sp[2].TS[2].WarnTsViolM : Last warning threshold value violation: minute / Dernier dépassement de la valeur seuil d'alarme : minute
   // Sp[2].TS[3].WarnTsViolM : Last warning threshold value violation: minute / Dernier dépassement de la valeur seuil d'alarme : minute
   // Sp[2].TS[4].WarnTsViolM : Last warning threshold value violation: minute / Dernier dépassement de la valeur seuil d'alarme : minute
   // Sp[2].TS[5].WarnTsViolM : Last warning threshold value violation: minute / Dernier dépassement de la valeur seuil d'alarme : minute
   // Sp[2].TS[6].WarnTsViolM : Last warning threshold value violation: minute / Dernier dépassement de la valeur seuil d'alarme : minute
   // Sp[1].TS[2].WarnTsViolS : Last warning threshold value violation: second / Dernier dépassement de la valeur seuil d'alarme : seconde
   // Sp[1].TS[3].WarnTsViolS : Last warning threshold value violation: second / Dernier dépassement de la valeur seuil d'alarme : seconde
   // Sp[1].TS[4].WarnTsViolS : Last warning threshold value violation: second / Dernier dépassement de la valeur seuil d'alarme : seconde
   // Sp[1].TS[5].WarnTsViolS : Last warning threshold value violation: second / Dernier dépassement de la valeur seuil d'alarme : seconde
   // Sp[1].TS[6].WarnTsViolS : Last warning threshold value violation: second / Dernier dépassement de la valeur seuil d'alarme : seconde
   // Sp[2].TS[1].WarnTsViolS : Last warning threshold value violation: second / Dernier dépassement de la valeur seuil d'alarme : seconde
   // Sp[2].TS[2].WarnTsViolS : Last warning threshold value violation: second / Dernier dépassement de la valeur seuil d'alarme : seconde
   // Sp[2].TS[3].WarnTsViolS : Last warning threshold value violation: second / Dernier dépassement de la valeur seuil d'alarme : seconde
   // Sp[2].TS[4].WarnTsViolS : Last warning threshold value violation: second / Dernier dépassement de la valeur seuil d'alarme : seconde
   // Sp[2].TS[5].WarnTsViolS : Last warning threshold value violation: second / Dernier dépassement de la valeur seuil d'alarme : seconde
   // Sp[2].TS[6].WarnTsViolS : Last warning threshold value violation: second / Dernier dépassement de la valeur seuil d'alarme : seconde
   // Sp[1].TS[2].WarnDurLimitViol : Duration of warning threshold value violations / Durée de dépassement de la valeur seuil d'alarme
   // Sp[1].TS[3].WarnDurLimitViol : Duration of warning threshold value violations / Durée de dépassement de la valeur seuil d'alarme
   // Sp[1].TS[4].WarnDurLimitViol : Duration of warning threshold value violations / Durée de dépassement de la valeur seuil d'alarme
   // Sp[1].TS[5].WarnDurLimitViol : Duration of warning threshold value violations / Durée de dépassement de la valeur seuil d'alarme
   // Sp[1].TS[6].WarnDurLimitViol : Duration of warning threshold value violations / Durée de dépassement de la valeur seuil d'alarme
   // Sp[2].TS[1].WarnDurLimitViol : Duration of warning threshold value violations / Durée de dépassement de la valeur seuil d'alarme
   // Sp[2].TS[2].WarnDurLimitViol : Duration of warning threshold value violations / Durée de dépassement de la valeur seuil d'alarme
   // Sp[2].TS[3].WarnDurLimitViol : Duration of warning threshold value violations / Durée de dépassement de la valeur seuil d'alarme
   // Sp[2].TS[4].WarnDurLimitViol : Duration of warning threshold value violations / Durée de dépassement de la valeur seuil d'alarme
   // Sp[2].TS[5].WarnDurLimitViol : Duration of warning threshold value violations / Durée de dépassement de la valeur seuil d'alarme
   // Sp[2].TS[6].WarnDurLimitViol : Duration of warning threshold value violations / Durée de dépassement de la valeur seuil d'alarme
   // Sp[1].TS[2].FaultThreshold : Temperature sensor fault threshold value [°C] / Sonde thermométrique valeur seuil de défaut
   // Sp[1].TS[3].FaultThreshold : Temperature sensor fault threshold value [°C] / Sonde thermométrique valeur seuil de défaut
   // Sp[1].TS[4].FaultThreshold : Temperature sensor fault threshold value [°C] / Sonde thermométrique valeur seuil de défaut
   // Sp[1].TS[5].FaultThreshold : Temperature sensor fault threshold value [°C] / Sonde thermométrique valeur seuil de défaut
   // Sp[1].TS[6].FaultThreshold : Temperature sensor fault threshold value [°C] / Sonde thermométrique valeur seuil de défaut
   // Sp[2].TS[1].FaultThreshold : Temperature sensor fault threshold value [°C] / Sonde thermométrique valeur seuil de défaut
   // Sp[2].TS[2].FaultThreshold : Temperature sensor fault threshold value [°C] / Sonde thermométrique valeur seuil de défaut
   // Sp[2].TS[3].FaultThreshold : Temperature sensor fault threshold value [°C] / Sonde thermométrique valeur seuil de défaut
   // Sp[2].TS[4].FaultThreshold : Temperature sensor fault threshold value [°C] / Sonde thermométrique valeur seuil de défaut
   // Sp[2].TS[5].FaultThreshold : Temperature sensor fault threshold value [°C] / Sonde thermométrique valeur seuil de défaut
   // Sp[2].TS[6].FaultThreshold : Temperature sensor fault threshold value [°C] / Sonde thermométrique valeur seuil de défaut
   // Sp[1].TS[2].FaultNumLimitViol : Number of fault threshold value violations / Nombre de dépassements de la valeur seuil de défaut
   // Sp[1].TS[3].FaultNumLimitViol : Number of fault threshold value violations / Nombre de dépassements de la valeur seuil de défaut
   // Sp[1].TS[4].FaultNumLimitViol : Number of fault threshold value violations / Nombre de dépassements de la valeur seuil de défaut
   // Sp[1].TS[5].FaultNumLimitViol : Number of fault threshold value violations / Nombre de dépassements de la valeur seuil de défaut
   // Sp[1].TS[6].FaultNumLimitViol : Number of fault threshold value violations / Nombre de dépassements de la valeur seuil de défaut
   // Sp[2].TS[1].FaultNumLimitViol : Number of fault threshold value violations / Nombre de dépassements de la valeur seuil de défaut
   // Sp[2].TS[2].FaultNumLimitViol : Number of fault threshold value violations / Nombre de dépassements de la valeur seuil de défaut
   // Sp[2].TS[3].FaultNumLimitViol : Number of fault threshold value violations / Nombre de dépassements de la valeur seuil de défaut
   // Sp[2].TS[4].FaultNumLimitViol : Number of fault threshold value violations / Nombre de dépassements de la valeur seuil de défaut
   // Sp[2].TS[5].FaultNumLimitViol : Number of fault threshold value violations / Nombre de dépassements de la valeur seuil de défaut
   // Sp[2].TS[6].FaultNumLimitViol : Number of fault threshold value violations / Nombre de dépassements de la valeur seuil de défaut
   // Sp[1].TS[2].FaultTsViolYY : Last fault threshold value violation: year / Dernier dépassement de la valeur seuil de défaut : année
   // Sp[1].TS[3].FaultTsViolYY : Last fault threshold value violation: year / Dernier dépassement de la valeur seuil de défaut : année
   // Sp[1].TS[4].FaultTsViolYY : Last fault threshold value violation: year / Dernier dépassement de la valeur seuil de défaut : année
   // Sp[1].TS[5].FaultTsViolYY : Last fault threshold value violation: year / Dernier dépassement de la valeur seuil de défaut : année
   // Sp[1].TS[6].FaultTsViolYY : Last fault threshold value violation: year / Dernier dépassement de la valeur seuil de défaut : année
   // Sp[2].TS[1].FaultTsViolYY : Last fault threshold value violation: year / Dernier dépassement de la valeur seuil de défaut : année
   // Sp[2].TS[2].FaultTsViolYY : Last fault threshold value violation: year / Dernier dépassement de la valeur seuil de défaut : année
   // Sp[2].TS[3].FaultTsViolYY : Last fault threshold value violation: year / Dernier dépassement de la valeur seuil de défaut : année
   // Sp[2].TS[4].FaultTsViolYY : Last fault threshold value violation: year / Dernier dépassement de la valeur seuil de défaut : année
   // Sp[2].TS[5].FaultTsViolYY : Last fault threshold value violation: year / Dernier dépassement de la valeur seuil de défaut : année
   // Sp[2].TS[6].FaultTsViolYY : Last fault threshold value violation: year / Dernier dépassement de la valeur seuil de défaut : année
   // Sp[1].TS[2].FaultTsViolMM : Last fault threshold value violation: month / Dernier dépassement de la valeur seuil de défaut : mois
   // Sp[1].TS[3].FaultTsViolMM : Last fault threshold value violation: month / Dernier dépassement de la valeur seuil de défaut : mois
   // Sp[1].TS[4].FaultTsViolMM : Last fault threshold value violation: month / Dernier dépassement de la valeur seuil de défaut : mois
   // Sp[1].TS[5].FaultTsViolMM : Last fault threshold value violation: month / Dernier dépassement de la valeur seuil de défaut : mois
   // Sp[1].TS[6].FaultTsViolMM : Last fault threshold value violation: month / Dernier dépassement de la valeur seuil de défaut : mois
   // Sp[2].TS[1].FaultTsViolMM : Last fault threshold value violation: month / Dernier dépassement de la valeur seuil de défaut : mois
   // Sp[2].TS[2].FaultTsViolMM : Last fault threshold value violation: month / Dernier dépassement de la valeur seuil de défaut : mois
   // Sp[2].TS[3].FaultTsViolMM : Last fault threshold value violation: month / Dernier dépassement de la valeur seuil de défaut : mois
   // Sp[2].TS[4].FaultTsViolMM : Last fault threshold value violation: month / Dernier dépassement de la valeur seuil de défaut : mois
   // Sp[2].TS[5].FaultTsViolMM : Last fault threshold value violation: month / Dernier dépassement de la valeur seuil de défaut : mois
   // Sp[2].TS[6].FaultTsViolMM : Last fault threshold value violation: month / Dernier dépassement de la valeur seuil de défaut : mois
   // Sp[1].TS[2].FaultTsViolDD : Last fault threshold value violation: day / Dernier dépassement de la valeur seuil de défaut : jour
   // Sp[1].TS[3].FaultTsViolDD : Last fault threshold value violation: day / Dernier dépassement de la valeur seuil de défaut : jour
   // Sp[1].TS[4].FaultTsViolDD : Last fault threshold value violation: day / Dernier dépassement de la valeur seuil de défaut : jour
   // Sp[1].TS[5].FaultTsViolDD : Last fault threshold value violation: day / Dernier dépassement de la valeur seuil de défaut : jour
   // Sp[1].TS[6].FaultTsViolDD : Last fault threshold value violation: day / Dernier dépassement de la valeur seuil de défaut : jour
   // Sp[2].TS[1].FaultTsViolDD : Last fault threshold value violation: day / Dernier dépassement de la valeur seuil de défaut : jour
   // Sp[2].TS[2].FaultTsViolDD : Last fault threshold value violation: day / Dernier dépassement de la valeur seuil de défaut : jour
   // Sp[2].TS[3].FaultTsViolDD : Last fault threshold value violation: day / Dernier dépassement de la valeur seuil de défaut : jour
   // Sp[2].TS[4].FaultTsViolDD : Last fault threshold value violation: day / Dernier dépassement de la valeur seuil de défaut : jour
   // Sp[2].TS[5].FaultTsViolDD : Last fault threshold value violation: day / Dernier dépassement de la valeur seuil de défaut : jour
   // Sp[2].TS[6].FaultTsViolDD : Last fault threshold value violation: day / Dernier dépassement de la valeur seuil de défaut : jour
   // Sp[1].TS[2].FaultTsViolH : Last fault threshold value violation: hour / Dernier dépassement de la valeur seuil de défaut : heure
   // Sp[1].TS[3].FaultTsViolH : Last fault threshold value violation: hour / Dernier dépassement de la valeur seuil de défaut : heure
   // Sp[1].TS[4].FaultTsViolH : Last fault threshold value violation: hour / Dernier dépassement de la valeur seuil de défaut : heure
   // Sp[1].TS[5].FaultTsViolH : Last fault threshold value violation: hour / Dernier dépassement de la valeur seuil de défaut : heure
   // Sp[1].TS[6].FaultTsViolH : Last fault threshold value violation: hour / Dernier dépassement de la valeur seuil de défaut : heure
   // Sp[2].TS[1].FaultTsViolH : Last fault threshold value violation: hour / Dernier dépassement de la valeur seuil de défaut : heure
   // Sp[2].TS[2].FaultTsViolH : Last fault threshold value violation: hour / Dernier dépassement de la valeur seuil de défaut : heure
   // Sp[2].TS[3].FaultTsViolH : Last fault threshold value violation: hour / Dernier dépassement de la valeur seuil de défaut : heure
   // Sp[2].TS[4].FaultTsViolH : Last fault threshold value violation: hour / Dernier dépassement de la valeur seuil de défaut : heure
   // Sp[2].TS[5].FaultTsViolH : Last fault threshold value violation: hour / Dernier dépassement de la valeur seuil de défaut : heure
   // Sp[2].TS[6].FaultTsViolH : Last fault threshold value violation: hour / Dernier dépassement de la valeur seuil de défaut : heure
   // Sp[1].TS[2].FaultTsViolM : Last fault threshold value violation: minute / Dernier dépassement de la valeur seuil de défaut : minute
   // Sp[1].TS[3].FaultTsViolM : Last fault threshold value violation: minute / Dernier dépassement de la valeur seuil de défaut : minute
   // Sp[1].TS[4].FaultTsViolM : Last fault threshold value violation: minute / Dernier dépassement de la valeur seuil de défaut : minute
   // Sp[1].TS[5].FaultTsViolM : Last fault threshold value violation: minute / Dernier dépassement de la valeur seuil de défaut : minute
   // Sp[1].TS[6].FaultTsViolM : Last fault threshold value violation: minute / Dernier dépassement de la valeur seuil de défaut : minute
   // Sp[2].TS[1].FaultTsViolM : Last fault threshold value violation: minute / Dernier dépassement de la valeur seuil de défaut : minute
   // Sp[2].TS[2].FaultTsViolM : Last fault threshold value violation: minute / Dernier dépassement de la valeur seuil de défaut : minute
   // Sp[2].TS[3].FaultTsViolM : Last fault threshold value violation: minute / Dernier dépassement de la valeur seuil de défaut : minute
   // Sp[2].TS[4].FaultTsViolM : Last fault threshold value violation: minute / Dernier dépassement de la valeur seuil de défaut : minute
   // Sp[2].TS[5].FaultTsViolM : Last fault threshold value violation: minute / Dernier dépassement de la valeur seuil de défaut : minute
   // Sp[2].TS[6].FaultTsViolM : Last fault threshold value violation: minute / Dernier dépassement de la valeur seuil de défaut : minute
   // Sp[1].TS[2].FaultTsViolS : Last fault threshold value violation: second / Dernier dépassement de la valeur seuil de défaut : seconde
   // Sp[1].TS[3].FaultTsViolS : Last fault threshold value violation: second / Dernier dépassement de la valeur seuil de défaut : seconde
   // Sp[1].TS[4].FaultTsViolS : Last fault threshold value violation: second / Dernier dépassement de la valeur seuil de défaut : seconde
   // Sp[1].TS[5].FaultTsViolS : Last fault threshold value violation: second / Dernier dépassement de la valeur seuil de défaut : seconde
   // Sp[1].TS[6].FaultTsViolS : Last fault threshold value violation: second / Dernier dépassement de la valeur seuil de défaut : seconde
   // Sp[2].TS[1].FaultTsViolS : Last fault threshold value violation: second / Dernier dépassement de la valeur seuil de défaut : seconde
   // Sp[2].TS[2].FaultTsViolS : Last fault threshold value violation: second / Dernier dépassement de la valeur seuil de défaut : seconde
   // Sp[2].TS[3].FaultTsViolS : Last fault threshold value violation: second / Dernier dépassement de la valeur seuil de défaut : seconde
   // Sp[2].TS[4].FaultTsViolS : Last fault threshold value violation: second / Dernier dépassement de la valeur seuil de défaut : seconde
   // Sp[2].TS[5].FaultTsViolS : Last fault threshold value violation: second / Dernier dépassement de la valeur seuil de défaut : seconde
   // Sp[2].TS[6].FaultTsViolS : Last fault threshold value violation: second / Dernier dépassement de la valeur seuil de défaut : seconde
   // Sp[1].TS[2].FaultDurLimitViol : Duration of fault threshold value violations / Durée de dépassement de la valeur seuil de défaut
   // Sp[1].TS[3].FaultDurLimitViol : Duration of fault threshold value violations / Durée de dépassement de la valeur seuil de défaut
   // Sp[1].TS[4].FaultDurLimitViol : Duration of fault threshold value violations / Durée de dépassement de la valeur seuil de défaut
   // Sp[1].TS[5].FaultDurLimitViol : Duration of fault threshold value violations / Durée de dépassement de la valeur seuil de défaut
   // Sp[1].TS[6].FaultDurLimitViol : Duration of fault threshold value violations / Durée de dépassement de la valeur seuil de défaut
   // Sp[2].TS[1].FaultDurLimitViol : Duration of fault threshold value violations / Durée de dépassement de la valeur seuil de défaut
   // Sp[2].TS[2].FaultDurLimitViol : Duration of fault threshold value violations / Durée de dépassement de la valeur seuil de défaut
   // Sp[2].TS[3].FaultDurLimitViol : Duration of fault threshold value violations / Durée de dépassement de la valeur seuil de défaut
   // Sp[2].TS[4].FaultDurLimitViol : Duration of fault threshold value violations / Durée de dépassement de la valeur seuil de défaut
   // Sp[2].TS[5].FaultDurLimitViol : Duration of fault threshold value violations / Durée de dépassement de la valeur seuil de défaut
   // Sp[2].TS[6].FaultDurLimitViol : Duration of fault threshold value violations / Durée de dépassement de la valeur seuil de défaut
   // Sp[1].TS[1] : Temperature sensor / Sonde thermométrique
   // Sp[1].TS[2] : Temperature sensor / Sonde thermométrique
   // Sp[1].TS[3] : Temperature sensor / Sonde thermométrique
   // Sp[1].TS[4] : Temperature sensor / Sonde thermométrique
   // Sp[1].TS[5] : Temperature sensor / Sonde thermométrique
   // Sp[1].TS[6] : Temperature sensor / Sonde thermométrique
   // Sp[2].TS[1] : Temperature sensor / Sonde thermométrique
   // Sp[2].TS[2] : Temperature sensor / Sonde thermométrique
   // Sp[2].TS[3] : Temperature sensor / Sonde thermométrique
   // Sp[2].TS[4] : Temperature sensor / Sonde thermométrique
   // Sp[2].TS[5] : Temperature sensor / Sonde thermométrique
   // Sp[2].TS[6] : Temperature sensor / Sonde thermométrique
   // Sp[2].TS : Temperature sensor / Sonde thermométrique
   // Sp[1] : Spindle / Broche
   // Sp[2] : Spindle / Broche
END_DATA_BLOCK

DATA_BLOCK "LBP_Internal1"   // DB25000
TITLE = Internal DB for basic program / DB interne pour programme de base
{ S7_Optimized_Access := 'TRUE' }
AUTHOR : SINUMERIK
FAMILY : SINUMERIK_ONE
VERSION : 6.24
// DB only for internal use in the basic program / DB réservé à l'utilisation interne dans le programme de base
// stored: IsWriteProtectedInAS true, MemoryReserve 100
   VAR
      McpCommIniData : Array[0..32] of Struct
         mcpType : Byte;
         mcpName : String;
         cycleMCPSend : Time;
         minMCPSend : Time;
         clientSendTimeout : Time;
         mcpSendTimeout : Time;
         mcpSendWarning : Time;
         cycleClientSend : Time;
         handwheelOption : Bool;
         paramDataLength : UInt;
         paramData : Array[1..5] of Byte;
         paramDataDckLength : UInt;
         paramDataDck : Array[1..5] of Byte;
      END_STRUCT;
      McpCommDomain : String := 'local.';
      McpCommMcp1 : Struct
         useIpAddress : Bool;
         ipAddress : Array[1..4] of USInt;
      END_STRUCT;
      McpCommMcp2 : Struct
         useIpAddress : Bool;
         ipAddress : Array[1..4] of USInt;
      END_STRUCT;
      McpCommHt : Struct
         useIpAddress : Bool;
         ipAddress : Array[1..4] of USInt;
      END_STRUCT;
      McpCommDck1 : Struct
         useIpAddress : Bool;
         ipAddress : Array[1..4] of USInt;
      END_STRUCT;
      McpCommDck2 : Struct
         useIpAddress : Bool;
         ipAddress : Array[1..4] of USInt;
      END_STRUCT;
      McpCommIdent : Struct
         useIpAddress : Bool;
         ipAddress : Array[1..4] of USInt;
      END_STRUCT;
   END_VAR
BEGIN
   McpCommIniData[0].mcpType := 16#0080;
   McpCommIniData[1].mcpType := 16#0081;
   McpCommIniData[2].mcpType := 16#0082;
   McpCommIniData[3].mcpType := 16#0083;
   McpCommIniData[4].mcpType := 16#0084;
   McpCommIniData[5].mcpType := 16#0085;
   McpCommIniData[6].mcpType := 16#0086;
   McpCommIniData[7].mcpType := 16#0087;
   McpCommIniData[8].mcpType := 16#0088;
   McpCommIniData[9].mcpType := 16#0089;
   McpCommIniData[10].mcpType := 16#008A;
   McpCommIniData[11].mcpType := 16#008B;
   McpCommIniData[12].mcpType := 16#008C;
   McpCommIniData[13].mcpType := 16#008D;
   McpCommIniData[14].mcpType := 16#008E;
   McpCommIniData[16].mcpType := 16#0090;
   McpCommIniData[17].mcpType := 16#0091;
   McpCommIniData[32].mcpType := 16#00A0;
   McpCommIniData[0].mcpName := 'MCP_483C';
   McpCommIniData[1].mcpName := 'MCP_483';
   McpCommIniData[2].mcpName := 'MCP_310';
   McpCommIniData[3].mcpName := 'MCP_OEM';
   McpCommIniData[4].mcpName := 'MCP_DMG';
   McpCommIniData[5].mcpName := 'HT_8';
   McpCommIniData[6].mcpName := 'TCU_DT';
   McpCommIniData[7].mcpName := 'MCP_MPP';
   McpCommIniData[8].mcpName := 'HT_2';
   McpCommIniData[9].mcpName := 'OP_08T';
   McpCommIniData[10].mcpName := 'MCP 310C PN';
   McpCommIniData[11].mcpName := 'MCP INDEX OEM';
   McpCommIniData[12].mcpName := 'RCU/TCU30';
   McpCommIniData[13].mcpName := 'MCP Interface PN';
   McpCommIniData[14].mcpName := 'VDCK';
   McpCommIniData[16].mcpName := 'MCP_398C';
   McpCommIniData[17].mcpName := 'HT_10';
   McpCommIniData[32].mcpName := 'MODULAR_MCP';
   McpCommIniData[0..7].cycleMCPSend := T#200MS;
   McpCommIniData[8].cycleMCPSend := T#50MS;
   McpCommIniData[9..14].cycleMCPSend := T#200MS;
   McpCommIniData[16].cycleMCPSend := T#200MS;
   McpCommIniData[17].cycleMCPSend := T#30MS;
   McpCommIniData[32].cycleMCPSend := T#30ms;
   McpCommIniData[0..5].minMCPSend := T#20MS;
   McpCommIniData[6].minMCPSend := T#50MS;
   McpCommIniData[7..8].minMCPSend := T#20MS;
   McpCommIniData[9].minMCPSend := T#50MS;
   McpCommIniData[10..11].minMCPSend := T#20MS;
   McpCommIniData[12].minMCPSend := T#50MS;
   McpCommIniData[13..14].minMCPSend := T#20MS;
   McpCommIniData[16].minMCPSend := T#20MS;
   McpCommIniData[17].minMCPSend := T#10MS;
   McpCommIniData[32].minMCPSend := T#10ms;
   McpCommIniData[0..13].clientSendTimeout := T#1S_500MS;
   McpCommIniData[14].clientSendTimeout := T#1S_200MS;
   McpCommIniData[16].clientSendTimeout := T#1S_500MS;
   McpCommIniData[17].clientSendTimeout := T#500MS;
   McpCommIniData[32].clientSendTimeout := T#500ms;
   McpCommIniData[0..13].mcpSendTimeout := T#1S_500MS;
   McpCommIniData[14].mcpSendTimeout := T#1S_200MS;
   McpCommIniData[16].mcpSendTimeout := T#1S_500MS;
   McpCommIniData[17].mcpSendTimeout := T#500MS;
   McpCommIniData[32].mcpSendTimeout := T#500ms;
   McpCommIniData[0..7].mcpSendWarning := T#600MS;
   McpCommIniData[8].mcpSendWarning := T#150MS;
   McpCommIniData[9..14].mcpSendWarning := T#600MS;
   McpCommIniData[16].mcpSendWarning := T#600MS;
   McpCommIniData[17].mcpSendWarning := T#200MS;
   McpCommIniData[32].mcpSendWarning := T#200ms;
   McpCommIniData[0..4].cycleClientSend := T#50MS;
   McpCommIniData[5..6].cycleClientSend := T#200MS;
   McpCommIniData[7..11].cycleClientSend := T#50MS;
   McpCommIniData[12].cycleClientSend := T#200MS;
   McpCommIniData[13].cycleClientSend := T#50MS;
   McpCommIniData[14].cycleClientSend := T#200MS;
   McpCommIniData[16].cycleClientSend := T#50MS;
   McpCommIniData[17].cycleClientSend := T#100MS;
   McpCommIniData[32].cycleClientSend := T#100ms;
   McpCommIniData[8].handwheelOption := true;
   McpCommIniData[0..5].paramDataLength := 5;
   McpCommIniData[6].paramDataLength := 3;
   McpCommIniData[7..8].paramDataLength := 5;
   McpCommIniData[9].paramDataLength := 3;
   McpCommIniData[10..11].paramDataLength := 5;
   McpCommIniData[12].paramDataLength := 3;
   McpCommIniData[13].paramDataLength := 5;
   McpCommIniData[14].paramDataLength := 3;
   McpCommIniData[16..17].paramDataLength := 5;
   McpCommIniData[32].paramDataLength := 2;
   McpCommIniData[0].paramData[1] := 16#0080;
   McpCommIniData[0].paramData[2] := 16#00C0;
   McpCommIniData[0].paramData[3] := 16#0007;
   McpCommIniData[0].paramData[4] := 16#000D;
   McpCommIniData[0].paramData[5] := 16#0051;
   McpCommIniData[1].paramData[1] := 16#0081;
   McpCommIniData[1].paramData[2] := 16#00C0;
   McpCommIniData[1].paramData[3] := 16#0007;
   McpCommIniData[1].paramData[4] := 16#000D;
   McpCommIniData[1].paramData[5] := 16#0051;
   McpCommIniData[2].paramData[1] := 16#0082;
   McpCommIniData[2].paramData[2] := 16#00C0;
   McpCommIniData[2].paramData[3] := 16#0007;
   McpCommIniData[2].paramData[4] := 16#000D;
   McpCommIniData[2].paramData[5] := 16#0051;
   McpCommIniData[3].paramData[1] := 16#0083;
   McpCommIniData[3].paramData[2] := 16#00C0;
   McpCommIniData[3].paramData[3] := 16#0007;
   McpCommIniData[3].paramData[4] := 16#000D;
   McpCommIniData[3].paramData[5] := 16#0051;
   McpCommIniData[4].paramData[1] := 16#0084;
   McpCommIniData[4].paramData[2] := 16#00C0;
   McpCommIniData[4].paramData[3] := 16#0009;
   McpCommIniData[4].paramData[4] := 16#000D;
   McpCommIniData[4].paramData[5] := 16#0051;
   McpCommIniData[5].paramData[1] := 16#0085;
   McpCommIniData[5].paramData[2] := 16#00C0;
   McpCommIniData[5].paramData[3..4] := 16#0007;
   McpCommIniData[5].paramData[5] := 16#0050;
   McpCommIniData[6].paramData[1] := 16#0086;
   McpCommIniData[6].paramData[2] := 16#0040;
   McpCommIniData[6].paramData[3] := 16#0001;
   McpCommIniData[7].paramData[1] := 16#0087;
   McpCommIniData[7].paramData[2] := 16#00C0;
   McpCommIniData[7].paramData[3] := 16#0007;
   McpCommIniData[7].paramData[4] := 16#000D;
   McpCommIniData[7].paramData[5] := 16#0051;
   McpCommIniData[8].paramData[1] := 16#0088;
   McpCommIniData[8].paramData[2] := 16#00C0;
   McpCommIniData[8].paramData[3] := 16#0013;
   McpCommIniData[8].paramData[4] := 16#0005;
   McpCommIniData[8].paramData[5] := 16#0050;
   McpCommIniData[9].paramData[1] := 16#0089;
   McpCommIniData[9].paramData[2] := 16#0040;
   McpCommIniData[9].paramData[3] := 16#0001;
   McpCommIniData[10].paramData[1] := 16#008A;
   McpCommIniData[10].paramData[2] := 16#00C0;
   McpCommIniData[10].paramData[3] := 16#0007;
   McpCommIniData[10].paramData[4] := 16#000D;
   McpCommIniData[10].paramData[5] := 16#0051;
   McpCommIniData[11].paramData[1] := 16#008B;
   McpCommIniData[11].paramData[2] := 16#00C0;
   McpCommIniData[11].paramData[3] := 16#0007;
   McpCommIniData[11].paramData[4] := 16#000D;
   McpCommIniData[11].paramData[5] := 16#0051;
   McpCommIniData[12].paramData[1] := 16#008C;
   McpCommIniData[12].paramData[2] := 16#0040;
   McpCommIniData[12].paramData[3] := 16#0001;
   McpCommIniData[13].paramData[1] := 16#008D;
   McpCommIniData[13].paramData[2] := 16#00C0;
   McpCommIniData[13].paramData[3] := 16#0009;
   McpCommIniData[13].paramData[4] := 16#000D;
   McpCommIniData[13].paramData[5] := 16#0051;
   McpCommIniData[14].paramData[1] := 16#008E;
   McpCommIniData[14].paramData[2] := 16#0040;
   McpCommIniData[14].paramData[3] := 16#0001;
   McpCommIniData[16].paramData[1] := 16#0090;
   McpCommIniData[16].paramData[2] := 16#00C0;
   McpCommIniData[16].paramData[3] := 16#0007;
   McpCommIniData[16].paramData[4] := 16#000D;
   McpCommIniData[16].paramData[5] := 16#0051;
   McpCommIniData[17].paramData[1] := 16#0091;
   McpCommIniData[17].paramData[2] := 16#00C0;
   McpCommIniData[17].paramData[3..4] := 16#0007;
   McpCommIniData[17].paramData[5] := 16#0050;
   McpCommIniData[32].paramData[1] := 16#A0;
   McpCommIniData[32].paramData[2] := 16#FF;
   McpCommIniData[1..7].paramDataDckLength := 3;
   McpCommIniData[9].paramDataDckLength := 3;
   McpCommIniData[12].paramDataDckLength := 3;
   McpCommIniData[14].paramDataDckLength := 3;
   McpCommIniData[17].paramDataDckLength := 3;
   McpCommIniData[32].paramDataDckLength := 2;
   McpCommIniData[1].paramDataDck[1] := 16#0081;
   McpCommIniData[1].paramDataDck[2] := 16#0040;
   McpCommIniData[1].paramDataDck[3] := 16#0001;
   McpCommIniData[2].paramDataDck[1] := 16#0082;
   McpCommIniData[2].paramDataDck[2] := 16#0040;
   McpCommIniData[2].paramDataDck[3] := 16#0001;
   McpCommIniData[3].paramDataDck[1] := 16#0083;
   McpCommIniData[3].paramDataDck[2] := 16#0040;
   McpCommIniData[3].paramDataDck[3] := 16#0001;
   McpCommIniData[4].paramDataDck[1] := 16#0084;
   McpCommIniData[4].paramDataDck[2] := 16#0040;
   McpCommIniData[4].paramDataDck[3] := 16#0001;
   McpCommIniData[5].paramDataDck[1] := 16#0085;
   McpCommIniData[5].paramDataDck[2] := 16#0040;
   McpCommIniData[5].paramDataDck[3] := 16#0001;
   McpCommIniData[6].paramDataDck[1] := 16#0086;
   McpCommIniData[6].paramDataDck[2] := 16#0040;
   McpCommIniData[6].paramDataDck[3] := 16#0001;
   McpCommIniData[7].paramDataDck[1] := 16#0087;
   McpCommIniData[7].paramDataDck[2] := 16#0040;
   McpCommIniData[7].paramDataDck[3] := 16#0001;
   McpCommIniData[9].paramDataDck[1] := 16#0089;
   McpCommIniData[9].paramDataDck[2] := 16#0040;
   McpCommIniData[9].paramDataDck[3] := 16#0001;
   McpCommIniData[12].paramDataDck[1] := 16#008C;
   McpCommIniData[12].paramDataDck[2] := 16#0040;
   McpCommIniData[12].paramDataDck[3] := 16#0001;
   McpCommIniData[14].paramDataDck[1] := 16#008E;
   McpCommIniData[14].paramDataDck[2] := 16#0040;
   McpCommIniData[14].paramDataDck[3] := 16#0001;
   McpCommIniData[17].paramDataDck[1] := 16#0091;
   McpCommIniData[17].paramDataDck[2] := 16#0040;
   McpCommIniData[17].paramDataDck[3] := 16#0001;
   McpCommIniData[32].paramDataDck[1] := 16#A0;
   McpCommIniData[32].paramDataDck[2] := 16#FF;
END_DATA_BLOCK

DATA_BLOCK "LBP_InternalDB25003"   // DB25003
TITLE = Internal DB for basic program / DB interne pour programme de base
{ S7_Optimized_Access := 'FALSE' }
AUTHOR : SINUMERIK
FAMILY : SINUMERIK_ONE
VERSION : 6.24
// DB only for internal use in the basic program / DB réservé à l'utilisation interne dans le programme de base
// stored: AutoNumber false
   VAR
      traceVar : Struct   // internal use only / réservé à l'utilisation interne
         cmdToPlc { ExternalVisible := 'False'} : Bool;
         identifier { ExternalVisible := 'False'} : UInt;
         symbol { ExternalVisible := 'False'} : WString;
         result { ExternalVisible := 'False'; ExternalWritable := 'False'} : UInt;
         unit { ExternalVisible := 'False'; ExternalWritable := 'False'} : UInt;
         column { ExternalVisible := 'False'; ExternalWritable := 'False'} : UInt;
         row { ExternalVisible := 'False'; ExternalWritable := 'False'} : UInt;
         "type" { ExternalVisible := 'False'; ExternalWritable := 'False'} : UInt;
      END_STRUCT;
   END_VAR
BEGIN
END_DATA_BLOCK

DATA_BLOCK "LBP_InternalDB8"   // DB8
TITLE = Internal DB for basic program / DB interne pour programme de base
{ S7_Optimized_Access := 'FALSE' }
AUTHOR : SINUMERIK
FAMILY : SINUMERIK_ONE
VERSION : 6.24
// DB only for internal use in the basic program / DB réservé à l'utilisation interne dans le programme de base
// stored: AutoNumber false
   VAR RETAIN
      DoNotUse0 : DWord;
      Reserved4 : Array[4..7] of Byte;
      FirstCycle : Byte;   // not used / non utilisé
      InternalUse9_0 : Bool;
      InternalUse9_1 : Bool;
      AL_404031 : Bool;
      InternalUse9_3 : Bool;
      InternalUse10 : Array[1..10] of Bool;
      InternalUse12 : SInt;
      InternalUse14 : Array[1..10] of Bool;
      InternalUse16 : SInt;
      InternalUse18 : Array[1..10] of Bool;
      InternalUse20 : Array[1..10] of Bool;
      Reserved22 : Array[22..53] of Byte;   // not used / non utilisé
      InternalUse54 : DWord;
      InternalUse58 : DWord;
      DoNotUse62 : DWord;
      Reserved66 : Array[66..75] of Byte;
      InternalUse76 : DWord;
      InternalUse80 : DInt;   // internal use only / réservé à l'utilisation interne
      InternalUse84 : LReal;   // internal use only / réservé à l'utilisation interne
      MinCycleTime : Int;   // not used / non utilisé
      AdaptTime : Int;   // not used / non utilisé
      ActCycleTime : Int;   // not used / non utilisé
      InternalUse98 : HW_ANY;   // internal use only / réservé à l'utilisation interne
      InternalUse100 : LReal;
   END_VAR
BEGIN
END_DATA_BLOCK

DATA_BLOCK "DB_NcVarSelect_AA_IM"   // DB63
{ S7_Optimized_Access := 'TRUE' }
// stored: MemoryReserve 100
   VAR
      "$AA_IM_Axis01_X" { S7_SetPoint := 'True'} : "LBP_typeNCVariableTokenLReal";
      "$AA_IM_Axis02_Y" { S7_SetPoint := 'True'} : "LBP_typeNCVariableTokenLReal";
      "$AA_IM_Axis03_ZM" { S7_SetPoint := 'True'} : "LBP_typeNCVariableTokenLReal";
      "$AA_IM_Axis04_B" { S7_SetPoint := 'True'} : "LBP_typeNCVariableTokenLReal";
      "$AA_IM_Axis05_U1" { S7_SetPoint := 'True'} : "LBP_typeNCVariableTokenLReal";
      "$AA_IM_Axis06_U2" { S7_SetPoint := 'True'} : "LBP_typeNCVariableTokenLReal";
      "$AA_IM_Axis07_V" { S7_SetPoint := 'True'} : "LBP_typeNCVariableTokenLReal";
      "$AA_IM_Axis08_W" { S7_SetPoint := 'True'} : "LBP_typeNCVariableTokenLReal";
      "$AA_IM_Axis09_ZL" { S7_SetPoint := 'True'} : "LBP_typeNCVariableTokenLReal";
   END_VAR
BEGIN
   "$AA_IM_Axis01_X".token.syntaxId := 16#82;
   "$AA_IM_Axis01_X".token.areaAndUnit := 16#41;
   "$AA_IM_Axis01_X".token.column := 16#2;
   "$AA_IM_Axis01_X".token.row := 16#1;
   "$AA_IM_Axis01_X".token.blockType := 16#74;
   "$AA_IM_Axis01_X".token.numberOfRows := 16#1;
   "$AA_IM_Axis01_X".token.dataTypeCode := 16#F;
   "$AA_IM_Axis01_X".token.length := 16#8;
   "$AA_IM_Axis02_Y".token.syntaxId := 16#82;
   "$AA_IM_Axis02_Y".token.areaAndUnit := 16#41;
   "$AA_IM_Axis02_Y".token.column := 16#2;
   "$AA_IM_Axis02_Y".token.row := 16#2;
   "$AA_IM_Axis02_Y".token.blockType := 16#74;
   "$AA_IM_Axis02_Y".token.numberOfRows := 16#1;
   "$AA_IM_Axis02_Y".token.dataTypeCode := 16#F;
   "$AA_IM_Axis02_Y".token.length := 16#8;
   "$AA_IM_Axis03_ZM".token.syntaxId := 16#82;
   "$AA_IM_Axis03_ZM".token.areaAndUnit := 16#41;
   "$AA_IM_Axis03_ZM".token.column := 16#2;
   "$AA_IM_Axis03_ZM".token.row := 16#3;
   "$AA_IM_Axis03_ZM".token.blockType := 16#74;
   "$AA_IM_Axis03_ZM".token.numberOfRows := 16#1;
   "$AA_IM_Axis03_ZM".token.dataTypeCode := 16#F;
   "$AA_IM_Axis03_ZM".token.length := 16#8;
   "$AA_IM_Axis04_B".token.syntaxId := 16#82;
   "$AA_IM_Axis04_B".token.areaAndUnit := 16#41;
   "$AA_IM_Axis04_B".token.column := 16#2;
   "$AA_IM_Axis04_B".token.row := 16#4;
   "$AA_IM_Axis04_B".token.blockType := 16#74;
   "$AA_IM_Axis04_B".token.numberOfRows := 16#1;
   "$AA_IM_Axis04_B".token.dataTypeCode := 16#F;
   "$AA_IM_Axis04_B".token.length := 16#8;
   "$AA_IM_Axis05_U1".token.syntaxId := 16#82;
   "$AA_IM_Axis05_U1".token.areaAndUnit := 16#41;
   "$AA_IM_Axis05_U1".token.column := 16#2;
   "$AA_IM_Axis05_U1".token.row := 16#5;
   "$AA_IM_Axis05_U1".token.blockType := 16#74;
   "$AA_IM_Axis05_U1".token.numberOfRows := 16#1;
   "$AA_IM_Axis05_U1".token.dataTypeCode := 16#F;
   "$AA_IM_Axis05_U1".token.length := 16#8;
   "$AA_IM_Axis06_U2".token.syntaxId := 16#82;
   "$AA_IM_Axis06_U2".token.areaAndUnit := 16#41;
   "$AA_IM_Axis06_U2".token.column := 16#2;
   "$AA_IM_Axis06_U2".token.row := 16#6;
   "$AA_IM_Axis06_U2".token.blockType := 16#74;
   "$AA_IM_Axis06_U2".token.numberOfRows := 16#1;
   "$AA_IM_Axis06_U2".token.dataTypeCode := 16#F;
   "$AA_IM_Axis06_U2".token.length := 16#8;
   "$AA_IM_Axis07_V".token.syntaxId := 16#82;
   "$AA_IM_Axis07_V".token.areaAndUnit := 16#41;
   "$AA_IM_Axis07_V".token.column := 16#2;
   "$AA_IM_Axis07_V".token.row := 16#7;
   "$AA_IM_Axis07_V".token.blockType := 16#74;
   "$AA_IM_Axis07_V".token.numberOfRows := 16#1;
   "$AA_IM_Axis07_V".token.dataTypeCode := 16#F;
   "$AA_IM_Axis07_V".token.length := 16#8;
   "$AA_IM_Axis08_W".token.syntaxId := 16#82;
   "$AA_IM_Axis08_W".token.areaAndUnit := 16#41;
   "$AA_IM_Axis08_W".token.column := 16#2;
   "$AA_IM_Axis08_W".token.row := 16#8;
   "$AA_IM_Axis08_W".token.blockType := 16#74;
   "$AA_IM_Axis08_W".token.numberOfRows := 16#1;
   "$AA_IM_Axis08_W".token.dataTypeCode := 16#F;
   "$AA_IM_Axis08_W".token.length := 16#8;
   "$AA_IM_Axis09_ZL".token.syntaxId := 16#82;
   "$AA_IM_Axis09_ZL".token.areaAndUnit := 16#41;
   "$AA_IM_Axis09_ZL".token.column := 16#2;
   "$AA_IM_Axis09_ZL".token.row := 16#9;
   "$AA_IM_Axis09_ZL".token.blockType := 16#74;
   "$AA_IM_Axis09_ZL".token.numberOfRows := 16#1;
   "$AA_IM_Axis09_ZL".token.dataTypeCode := 16#F;
   "$AA_IM_Axis09_ZL".token.length := 16#8;
END_DATA_BLOCK

DATA_BLOCK "DB_NcVarSelect_MA_JOG_VELO"   // DB85
{ S7_Optimized_Access := 'TRUE' }
// stored: MemoryReserve 100
   VAR
      "$MA_JOG_VELO_Axis01_X" { S7_SetPoint := 'True'} : "LBP_typeNCVariableTokenLReal";
      "$MA_JOG_VELO_Axis02_Y" { S7_SetPoint := 'True'} : "LBP_typeNCVariableTokenLReal";
      "$MA_JOG_VELO_Axis03_ZM" { S7_SetPoint := 'True'} : "LBP_typeNCVariableTokenLReal";
      "$MA_JOG_VELO_Axis04_B" { S7_SetPoint := 'True'} : "LBP_typeNCVariableTokenLReal";
      "$MA_JOG_VELO_Axis05_U1" { S7_SetPoint := 'True'} : "LBP_typeNCVariableTokenLReal";
      "$MA_JOG_VELO_Axis06_U2" { S7_SetPoint := 'True'} : "LBP_typeNCVariableTokenLReal";
      "$MA_JOG_VELO_Axis07_V" { S7_SetPoint := 'True'} : "LBP_typeNCVariableTokenLReal";
      "$MA_JOG_VELO_Axis08_W" { S7_SetPoint := 'True'} : "LBP_typeNCVariableTokenLReal";
      "$MA_JOG_VELO_Axis09_ZL" { S7_SetPoint := 'True'} : "LBP_typeNCVariableTokenLReal";
   END_VAR
BEGIN
   "$MA_JOG_VELO_Axis01_X".token.syntaxId := 16#82;
   "$MA_JOG_VELO_Axis01_X".token.areaAndUnit := 16#61;
   "$MA_JOG_VELO_Axis01_X".token.column := 16#7D14;
   "$MA_JOG_VELO_Axis01_X".token.row := 16#1;
   "$MA_JOG_VELO_Axis01_X".token.blockType := 16#1A;
   "$MA_JOG_VELO_Axis01_X".token.numberOfRows := 16#1;
   "$MA_JOG_VELO_Axis01_X".token.dataTypeCode := 16#F;
   "$MA_JOG_VELO_Axis01_X".token.length := 16#8;
   "$MA_JOG_VELO_Axis02_Y".token.syntaxId := 16#82;
   "$MA_JOG_VELO_Axis02_Y".token.areaAndUnit := 16#62;
   "$MA_JOG_VELO_Axis02_Y".token.column := 16#7D14;
   "$MA_JOG_VELO_Axis02_Y".token.row := 16#1;
   "$MA_JOG_VELO_Axis02_Y".token.blockType := 16#1A;
   "$MA_JOG_VELO_Axis02_Y".token.numberOfRows := 16#1;
   "$MA_JOG_VELO_Axis02_Y".token.dataTypeCode := 16#F;
   "$MA_JOG_VELO_Axis02_Y".token.length := 16#8;
   "$MA_JOG_VELO_Axis03_ZM".token.syntaxId := 16#82;
   "$MA_JOG_VELO_Axis03_ZM".token.areaAndUnit := 16#63;
   "$MA_JOG_VELO_Axis03_ZM".token.column := 16#7D14;
   "$MA_JOG_VELO_Axis03_ZM".token.row := 16#1;
   "$MA_JOG_VELO_Axis03_ZM".token.blockType := 16#1A;
   "$MA_JOG_VELO_Axis03_ZM".token.numberOfRows := 16#1;
   "$MA_JOG_VELO_Axis03_ZM".token.dataTypeCode := 16#F;
   "$MA_JOG_VELO_Axis03_ZM".token.length := 16#8;
   "$MA_JOG_VELO_Axis04_B".token.syntaxId := 16#82;
   "$MA_JOG_VELO_Axis04_B".token.areaAndUnit := 16#64;
   "$MA_JOG_VELO_Axis04_B".token.column := 16#7D14;
   "$MA_JOG_VELO_Axis04_B".token.row := 16#1;
   "$MA_JOG_VELO_Axis04_B".token.blockType := 16#1A;
   "$MA_JOG_VELO_Axis04_B".token.numberOfRows := 16#1;
   "$MA_JOG_VELO_Axis04_B".token.dataTypeCode := 16#F;
   "$MA_JOG_VELO_Axis04_B".token.length := 16#8;
   "$MA_JOG_VELO_Axis05_U1".token.syntaxId := 16#82;
   "$MA_JOG_VELO_Axis05_U1".token.areaAndUnit := 16#65;
   "$MA_JOG_VELO_Axis05_U1".token.column := 16#7D14;
   "$MA_JOG_VELO_Axis05_U1".token.row := 16#1;
   "$MA_JOG_VELO_Axis05_U1".token.blockType := 16#1A;
   "$MA_JOG_VELO_Axis05_U1".token.numberOfRows := 16#1;
   "$MA_JOG_VELO_Axis05_U1".token.dataTypeCode := 16#F;
   "$MA_JOG_VELO_Axis05_U1".token.length := 16#8;
   "$MA_JOG_VELO_Axis06_U2".token.syntaxId := 16#82;
   "$MA_JOG_VELO_Axis06_U2".token.areaAndUnit := 16#66;
   "$MA_JOG_VELO_Axis06_U2".token.column := 16#7D14;
   "$MA_JOG_VELO_Axis06_U2".token.row := 16#1;
   "$MA_JOG_VELO_Axis06_U2".token.blockType := 16#1A;
   "$MA_JOG_VELO_Axis06_U2".token.numberOfRows := 16#1;
   "$MA_JOG_VELO_Axis06_U2".token.dataTypeCode := 16#F;
   "$MA_JOG_VELO_Axis06_U2".token.length := 16#8;
   "$MA_JOG_VELO_Axis07_V".token.syntaxId := 16#82;
   "$MA_JOG_VELO_Axis07_V".token.areaAndUnit := 16#67;
   "$MA_JOG_VELO_Axis07_V".token.column := 16#7D14;
   "$MA_JOG_VELO_Axis07_V".token.row := 16#1;
   "$MA_JOG_VELO_Axis07_V".token.blockType := 16#1A;
   "$MA_JOG_VELO_Axis07_V".token.numberOfRows := 16#1;
   "$MA_JOG_VELO_Axis07_V".token.dataTypeCode := 16#F;
   "$MA_JOG_VELO_Axis07_V".token.length := 16#8;
   "$MA_JOG_VELO_Axis08_W".token.syntaxId := 16#82;
   "$MA_JOG_VELO_Axis08_W".token.areaAndUnit := 16#68;
   "$MA_JOG_VELO_Axis08_W".token.column := 16#7D14;
   "$MA_JOG_VELO_Axis08_W".token.row := 16#1;
   "$MA_JOG_VELO_Axis08_W".token.blockType := 16#1A;
   "$MA_JOG_VELO_Axis08_W".token.numberOfRows := 16#1;
   "$MA_JOG_VELO_Axis08_W".token.dataTypeCode := 16#F;
   "$MA_JOG_VELO_Axis08_W".token.length := 16#8;
   "$MA_JOG_VELO_Axis09_ZL".token.syntaxId := 16#82;
   "$MA_JOG_VELO_Axis09_ZL".token.areaAndUnit := 16#69;
   "$MA_JOG_VELO_Axis09_ZL".token.column := 16#7D14;
   "$MA_JOG_VELO_Axis09_ZL".token.row := 16#1;
   "$MA_JOG_VELO_Axis09_ZL".token.blockType := 16#1A;
   "$MA_JOG_VELO_Axis09_ZL".token.numberOfRows := 16#1;
   "$MA_JOG_VELO_Axis09_ZL".token.dataTypeCode := 16#F;
   "$MA_JOG_VELO_Axis09_ZL".token.length := 16#8;
END_DATA_BLOCK

DATA_BLOCK "DB_NcVarSelect_MA_JOG_VELO_RAPID"   // DB65
{ S7_Optimized_Access := 'TRUE' }
// stored: MemoryReserve 100
   VAR
      "$MA_JOG_VELO_RAPID_Axis01_X" { S7_SetPoint := 'True'} : "LBP_typeNCVariableTokenLReal";
      "$MA_JOG_VELO_RAPID_Axis02_Y" { S7_SetPoint := 'True'} : "LBP_typeNCVariableTokenLReal";
      "$MA_JOG_VELO_RAPID_Axis03_ZM" { S7_SetPoint := 'True'} : "LBP_typeNCVariableTokenLReal";
      "$MA_JOG_VELO_RAPID_Axis04_B" { S7_SetPoint := 'True'} : "LBP_typeNCVariableTokenLReal";
      "$MA_JOG_VELO_RAPID_Axis05_U1" { S7_SetPoint := 'True'} : "LBP_typeNCVariableTokenLReal";
      "$MA_JOG_VELO_RAPID_Axis06_U2" { S7_SetPoint := 'True'} : "LBP_typeNCVariableTokenLReal";
      "$MA_JOG_VELO_RAPID_Axis07_V" { S7_SetPoint := 'True'} : "LBP_typeNCVariableTokenLReal";
      "$MA_JOG_VELO_RAPID_Axis08_W" { S7_SetPoint := 'True'} : "LBP_typeNCVariableTokenLReal";
      "$MA_JOG_VELO_RAPID_Axis09_ZL" { S7_SetPoint := 'True'} : "LBP_typeNCVariableTokenLReal";
   END_VAR
BEGIN
   "$MA_JOG_VELO_RAPID_Axis01_X".token.syntaxId := 16#82;
   "$MA_JOG_VELO_RAPID_Axis01_X".token.areaAndUnit := 16#61;
   "$MA_JOG_VELO_RAPID_Axis01_X".token.column := 16#7D0A;
   "$MA_JOG_VELO_RAPID_Axis01_X".token.row := 16#1;
   "$MA_JOG_VELO_RAPID_Axis01_X".token.blockType := 16#1A;
   "$MA_JOG_VELO_RAPID_Axis01_X".token.numberOfRows := 16#1;
   "$MA_JOG_VELO_RAPID_Axis01_X".token.dataTypeCode := 16#F;
   "$MA_JOG_VELO_RAPID_Axis01_X".token.length := 16#8;
   "$MA_JOG_VELO_RAPID_Axis02_Y".token.syntaxId := 16#82;
   "$MA_JOG_VELO_RAPID_Axis02_Y".token.areaAndUnit := 16#62;
   "$MA_JOG_VELO_RAPID_Axis02_Y".token.column := 16#7D0A;
   "$MA_JOG_VELO_RAPID_Axis02_Y".token.row := 16#1;
   "$MA_JOG_VELO_RAPID_Axis02_Y".token.blockType := 16#1A;
   "$MA_JOG_VELO_RAPID_Axis02_Y".token.numberOfRows := 16#1;
   "$MA_JOG_VELO_RAPID_Axis02_Y".token.dataTypeCode := 16#F;
   "$MA_JOG_VELO_RAPID_Axis02_Y".token.length := 16#8;
   "$MA_JOG_VELO_RAPID_Axis03_ZM".token.syntaxId := 16#82;
   "$MA_JOG_VELO_RAPID_Axis03_ZM".token.areaAndUnit := 16#63;
   "$MA_JOG_VELO_RAPID_Axis03_ZM".token.column := 16#7D0A;
   "$MA_JOG_VELO_RAPID_Axis03_ZM".token.row := 16#1;
   "$MA_JOG_VELO_RAPID_Axis03_ZM".token.blockType := 16#1A;
   "$MA_JOG_VELO_RAPID_Axis03_ZM".token.numberOfRows := 16#1;
   "$MA_JOG_VELO_RAPID_Axis03_ZM".token.dataTypeCode := 16#F;
   "$MA_JOG_VELO_RAPID_Axis03_ZM".token.length := 16#8;
   "$MA_JOG_VELO_RAPID_Axis04_B".token.syntaxId := 16#82;
   "$MA_JOG_VELO_RAPID_Axis04_B".token.areaAndUnit := 16#64;
   "$MA_JOG_VELO_RAPID_Axis04_B".token.column := 16#7D0A;
   "$MA_JOG_VELO_RAPID_Axis04_B".token.row := 16#1;
   "$MA_JOG_VELO_RAPID_Axis04_B".token.blockType := 16#1A;
   "$MA_JOG_VELO_RAPID_Axis04_B".token.numberOfRows := 16#1;
   "$MA_JOG_VELO_RAPID_Axis04_B".token.dataTypeCode := 16#F;
   "$MA_JOG_VELO_RAPID_Axis04_B".token.length := 16#8;
   "$MA_JOG_VELO_RAPID_Axis05_U1".token.syntaxId := 16#82;
   "$MA_JOG_VELO_RAPID_Axis05_U1".token.areaAndUnit := 16#65;
   "$MA_JOG_VELO_RAPID_Axis05_U1".token.column := 16#7D0A;
   "$MA_JOG_VELO_RAPID_Axis05_U1".token.row := 16#1;
   "$MA_JOG_VELO_RAPID_Axis05_U1".token.blockType := 16#1A;
   "$MA_JOG_VELO_RAPID_Axis05_U1".token.numberOfRows := 16#1;
   "$MA_JOG_VELO_RAPID_Axis05_U1".token.dataTypeCode := 16#F;
   "$MA_JOG_VELO_RAPID_Axis05_U1".token.length := 16#8;
   "$MA_JOG_VELO_RAPID_Axis06_U2".token.syntaxId := 16#82;
   "$MA_JOG_VELO_RAPID_Axis06_U2".token.areaAndUnit := 16#66;
   "$MA_JOG_VELO_RAPID_Axis06_U2".token.column := 16#7D0A;
   "$MA_JOG_VELO_RAPID_Axis06_U2".token.row := 16#1;
   "$MA_JOG_VELO_RAPID_Axis06_U2".token.blockType := 16#1A;
   "$MA_JOG_VELO_RAPID_Axis06_U2".token.numberOfRows := 16#1;
   "$MA_JOG_VELO_RAPID_Axis06_U2".token.dataTypeCode := 16#F;
   "$MA_JOG_VELO_RAPID_Axis06_U2".token.length := 16#8;
   "$MA_JOG_VELO_RAPID_Axis07_V".token.syntaxId := 16#82;
   "$MA_JOG_VELO_RAPID_Axis07_V".token.areaAndUnit := 16#67;
   "$MA_JOG_VELO_RAPID_Axis07_V".token.column := 16#7D0A;
   "$MA_JOG_VELO_RAPID_Axis07_V".token.row := 16#1;
   "$MA_JOG_VELO_RAPID_Axis07_V".token.blockType := 16#1A;
   "$MA_JOG_VELO_RAPID_Axis07_V".token.numberOfRows := 16#1;
   "$MA_JOG_VELO_RAPID_Axis07_V".token.dataTypeCode := 16#F;
   "$MA_JOG_VELO_RAPID_Axis07_V".token.length := 16#8;
   "$MA_JOG_VELO_RAPID_Axis08_W".token.syntaxId := 16#82;
   "$MA_JOG_VELO_RAPID_Axis08_W".token.areaAndUnit := 16#68;
   "$MA_JOG_VELO_RAPID_Axis08_W".token.column := 16#7D0A;
   "$MA_JOG_VELO_RAPID_Axis08_W".token.row := 16#1;
   "$MA_JOG_VELO_RAPID_Axis08_W".token.blockType := 16#1A;
   "$MA_JOG_VELO_RAPID_Axis08_W".token.numberOfRows := 16#1;
   "$MA_JOG_VELO_RAPID_Axis08_W".token.dataTypeCode := 16#F;
   "$MA_JOG_VELO_RAPID_Axis08_W".token.length := 16#8;
   "$MA_JOG_VELO_RAPID_Axis09_ZL".token.syntaxId := 16#82;
   "$MA_JOG_VELO_RAPID_Axis09_ZL".token.areaAndUnit := 16#69;
   "$MA_JOG_VELO_RAPID_Axis09_ZL".token.column := 16#7D0A;
   "$MA_JOG_VELO_RAPID_Axis09_ZL".token.row := 16#1;
   "$MA_JOG_VELO_RAPID_Axis09_ZL".token.blockType := 16#1A;
   "$MA_JOG_VELO_RAPID_Axis09_ZL".token.numberOfRows := 16#1;
   "$MA_JOG_VELO_RAPID_Axis09_ZL".token.dataTypeCode := 16#F;
   "$MA_JOG_VELO_RAPID_Axis09_ZL".token.length := 16#8;
END_DATA_BLOCK

DATA_BLOCK "DB_NcVarSelect_MA_POS_LIMIT_MINUS"   // DB66
{ S7_Optimized_Access := 'TRUE' }
// stored: MemoryReserve 100
   VAR
      "$MA_POS_LIMIT_MINUS_Axis01_X" { S7_SetPoint := 'True'} : "LBP_typeNCVariableTokenLReal";
      "$MA_POS_LIMIT_MINUS_Axis02_Y" { S7_SetPoint := 'True'} : "LBP_typeNCVariableTokenLReal";
      "$MA_POS_LIMIT_MINUS_Axis03_ZM" { S7_SetPoint := 'True'} : "LBP_typeNCVariableTokenLReal";
      "$MA_POS_LIMIT_MINUS_Axis04_B" { S7_SetPoint := 'True'} : "LBP_typeNCVariableTokenLReal";
      "$MA_POS_LIMIT_MINUS_Axis05_U1" { S7_SetPoint := 'True'} : "LBP_typeNCVariableTokenLReal";
      "$MA_POS_LIMIT_MINUS_Axis06_U2" { S7_SetPoint := 'True'} : "LBP_typeNCVariableTokenLReal";
      "$MA_POS_LIMIT_MINUS_Axis07_V" { S7_SetPoint := 'True'} : "LBP_typeNCVariableTokenLReal";
      "$MA_POS_LIMIT_MINUS_Axis08_W" { S7_SetPoint := 'True'} : "LBP_typeNCVariableTokenLReal";
      "$MA_POS_LIMIT_MINUS_Axis09_ZL" { S7_SetPoint := 'True'} : "LBP_typeNCVariableTokenLReal";
   END_VAR
BEGIN
   "$MA_POS_LIMIT_MINUS_Axis01_X".token.syntaxId := 16#82;
   "$MA_POS_LIMIT_MINUS_Axis01_X".token.areaAndUnit := 16#61;
   "$MA_POS_LIMIT_MINUS_Axis01_X".token.column := 16#8D04;
   "$MA_POS_LIMIT_MINUS_Axis01_X".token.row := 16#1;
   "$MA_POS_LIMIT_MINUS_Axis01_X".token.blockType := 16#1A;
   "$MA_POS_LIMIT_MINUS_Axis01_X".token.numberOfRows := 16#1;
   "$MA_POS_LIMIT_MINUS_Axis01_X".token.dataTypeCode := 16#F;
   "$MA_POS_LIMIT_MINUS_Axis01_X".token.length := 16#8;
   "$MA_POS_LIMIT_MINUS_Axis02_Y".token.syntaxId := 16#82;
   "$MA_POS_LIMIT_MINUS_Axis02_Y".token.areaAndUnit := 16#62;
   "$MA_POS_LIMIT_MINUS_Axis02_Y".token.column := 16#8D04;
   "$MA_POS_LIMIT_MINUS_Axis02_Y".token.row := 16#1;
   "$MA_POS_LIMIT_MINUS_Axis02_Y".token.blockType := 16#1A;
   "$MA_POS_LIMIT_MINUS_Axis02_Y".token.numberOfRows := 16#1;
   "$MA_POS_LIMIT_MINUS_Axis02_Y".token.dataTypeCode := 16#F;
   "$MA_POS_LIMIT_MINUS_Axis02_Y".token.length := 16#8;
   "$MA_POS_LIMIT_MINUS_Axis03_ZM".token.syntaxId := 16#82;
   "$MA_POS_LIMIT_MINUS_Axis03_ZM".token.areaAndUnit := 16#63;
   "$MA_POS_LIMIT_MINUS_Axis03_ZM".token.column := 16#8D04;
   "$MA_POS_LIMIT_MINUS_Axis03_ZM".token.row := 16#1;
   "$MA_POS_LIMIT_MINUS_Axis03_ZM".token.blockType := 16#1A;
   "$MA_POS_LIMIT_MINUS_Axis03_ZM".token.numberOfRows := 16#1;
   "$MA_POS_LIMIT_MINUS_Axis03_ZM".token.dataTypeCode := 16#F;
   "$MA_POS_LIMIT_MINUS_Axis03_ZM".token.length := 16#8;
   "$MA_POS_LIMIT_MINUS_Axis04_B".token.syntaxId := 16#82;
   "$MA_POS_LIMIT_MINUS_Axis04_B".token.areaAndUnit := 16#64;
   "$MA_POS_LIMIT_MINUS_Axis04_B".token.column := 16#8D04;
   "$MA_POS_LIMIT_MINUS_Axis04_B".token.row := 16#1;
   "$MA_POS_LIMIT_MINUS_Axis04_B".token.blockType := 16#1A;
   "$MA_POS_LIMIT_MINUS_Axis04_B".token.numberOfRows := 16#1;
   "$MA_POS_LIMIT_MINUS_Axis04_B".token.dataTypeCode := 16#F;
   "$MA_POS_LIMIT_MINUS_Axis04_B".token.length := 16#8;
   "$MA_POS_LIMIT_MINUS_Axis05_U1".token.syntaxId := 16#82;
   "$MA_POS_LIMIT_MINUS_Axis05_U1".token.areaAndUnit := 16#65;
   "$MA_POS_LIMIT_MINUS_Axis05_U1".token.column := 16#8D04;
   "$MA_POS_LIMIT_MINUS_Axis05_U1".token.row := 16#1;
   "$MA_POS_LIMIT_MINUS_Axis05_U1".token.blockType := 16#1A;
   "$MA_POS_LIMIT_MINUS_Axis05_U1".token.numberOfRows := 16#1;
   "$MA_POS_LIMIT_MINUS_Axis05_U1".token.dataTypeCode := 16#F;
   "$MA_POS_LIMIT_MINUS_Axis05_U1".token.length := 16#8;
   "$MA_POS_LIMIT_MINUS_Axis06_U2".token.syntaxId := 16#82;
   "$MA_POS_LIMIT_MINUS_Axis06_U2".token.areaAndUnit := 16#66;
   "$MA_POS_LIMIT_MINUS_Axis06_U2".token.column := 16#8D04;
   "$MA_POS_LIMIT_MINUS_Axis06_U2".token.row := 16#1;
   "$MA_POS_LIMIT_MINUS_Axis06_U2".token.blockType := 16#1A;
   "$MA_POS_LIMIT_MINUS_Axis06_U2".token.numberOfRows := 16#1;
   "$MA_POS_LIMIT_MINUS_Axis06_U2".token.dataTypeCode := 16#F;
   "$MA_POS_LIMIT_MINUS_Axis06_U2".token.length := 16#8;
   "$MA_POS_LIMIT_MINUS_Axis07_V".token.syntaxId := 16#82;
   "$MA_POS_LIMIT_MINUS_Axis07_V".token.areaAndUnit := 16#67;
   "$MA_POS_LIMIT_MINUS_Axis07_V".token.column := 16#8D04;
   "$MA_POS_LIMIT_MINUS_Axis07_V".token.row := 16#1;
   "$MA_POS_LIMIT_MINUS_Axis07_V".token.blockType := 16#1A;
   "$MA_POS_LIMIT_MINUS_Axis07_V".token.numberOfRows := 16#1;
   "$MA_POS_LIMIT_MINUS_Axis07_V".token.dataTypeCode := 16#F;
   "$MA_POS_LIMIT_MINUS_Axis07_V".token.length := 16#8;
   "$MA_POS_LIMIT_MINUS_Axis08_W".token.syntaxId := 16#82;
   "$MA_POS_LIMIT_MINUS_Axis08_W".token.areaAndUnit := 16#68;
   "$MA_POS_LIMIT_MINUS_Axis08_W".token.column := 16#8D04;
   "$MA_POS_LIMIT_MINUS_Axis08_W".token.row := 16#1;
   "$MA_POS_LIMIT_MINUS_Axis08_W".token.blockType := 16#1A;
   "$MA_POS_LIMIT_MINUS_Axis08_W".token.numberOfRows := 16#1;
   "$MA_POS_LIMIT_MINUS_Axis08_W".token.dataTypeCode := 16#F;
   "$MA_POS_LIMIT_MINUS_Axis08_W".token.length := 16#8;
   "$MA_POS_LIMIT_MINUS_Axis09_ZL".token.syntaxId := 16#82;
   "$MA_POS_LIMIT_MINUS_Axis09_ZL".token.areaAndUnit := 16#69;
   "$MA_POS_LIMIT_MINUS_Axis09_ZL".token.column := 16#8D04;
   "$MA_POS_LIMIT_MINUS_Axis09_ZL".token.row := 16#1;
   "$MA_POS_LIMIT_MINUS_Axis09_ZL".token.blockType := 16#1A;
   "$MA_POS_LIMIT_MINUS_Axis09_ZL".token.numberOfRows := 16#1;
   "$MA_POS_LIMIT_MINUS_Axis09_ZL".token.dataTypeCode := 16#F;
   "$MA_POS_LIMIT_MINUS_Axis09_ZL".token.length := 16#8;
END_DATA_BLOCK

